% RSLogix 500 project TASTEFULL SELECTIONBINSCRUBBER INDEXER AND UN-STACKER 2-08-2017.RSS, saved by version 10.00.00.00 %
PROJECT "TASTEFUL"    % processor: MicroLogix 1400 %

PROGRAM FILES
  LAD 2 "MAIN"  12 rungs
  LAD 3 "START/MODE"  12 rungs
  LAD 4 "ENCODER"  11 rungs
  LAD 5 "CRADLE"  26 rungs
  LAD 6 "BRUSH"  10 rungs
  LAD 7 "H20 TANKS"  26 rungs
  LAD 8 "AUXILARY"  4 rungs
  LAD 9 "FAULTS"  36 rungs
  LAD 10 "SPARE"  2 rungs
  LAD 11 "STAGING"  8 rungs
  LAD 12 "DESTACK LS"  19 rungs
  LAD 13 "DESTACK"  29 rungs

DATA FILES
  O0 OUTPUT  8 elements
  I1 INPUT  11 elements
  S2 STATUS  66 elements
  B3 BINARY  7 elements
  T4 TIMER  38 elements
  C5 COUNTER  1 elements
  R6 CONTROL  1 elements
  N7 INTEGER  40 elements
  F8 FLOAT  30 elements
  L9   1 elements
  L10   2 elements

LADDER 2 "MAIN"
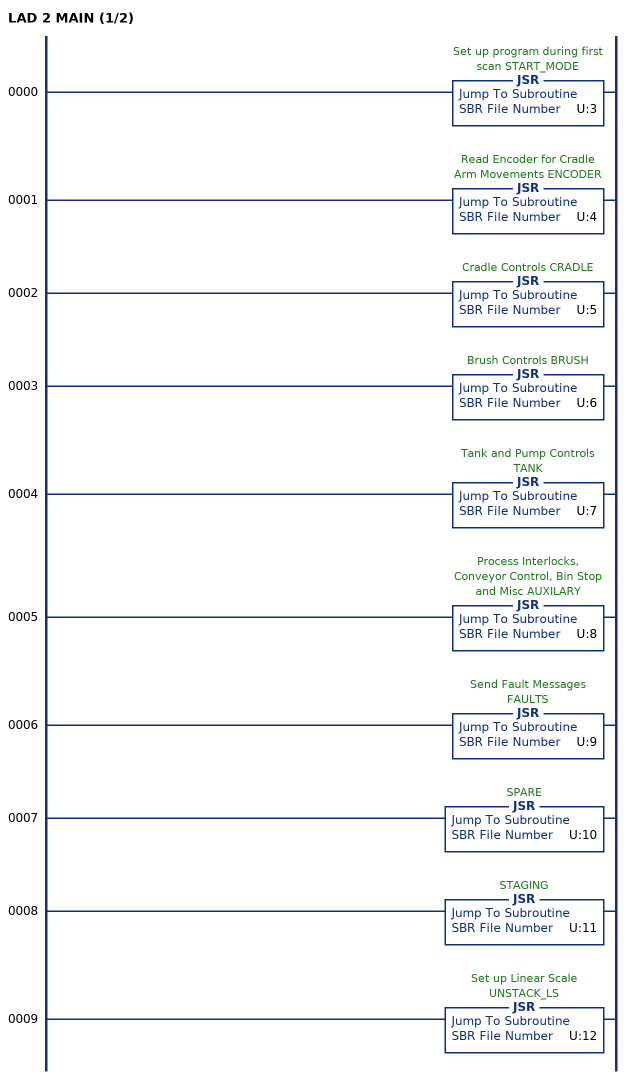
% Rung: 0 %
SOR JSR U:3 EOR
%   U:3  START_MODE  "Set up program during first scan" %
% Rung: 1 %
SOR JSR U:4 EOR
%   U:4  ENCODER  "Read Encoder for Cradle Arm Movements" %
% Rung: 2 %
SOR JSR U:5 EOR
%   U:5  CRADLE  "Cradle Controls" %
% Rung: 3 %
SOR JSR U:6 EOR
%   U:6  BRUSH  "Brush Controls" %
% Rung: 4 %
SOR JSR U:7 EOR
%   U:7  TANK  "Tank and Pump Controls" %
% Rung: 5 %
SOR JSR U:8 EOR
%   U:8  AUXILARY  "Process Interlocks, Conveyor Control, Bin Stop and Misc" %
% Rung: 6 %
SOR JSR U:9 EOR
%   U:9  FAULTS  "Send Fault Messages" %
% Rung: 7 %
SOR JSR U:10 EOR
%   U:10  SPARE %
% Rung: 8 %
SOR JSR U:11 EOR
%   U:11  STAGING %
% Rung: 9 %
SOR JSR U:12 EOR
%   U:12  UNSTACK_LS  "Set up Linear Scale" %

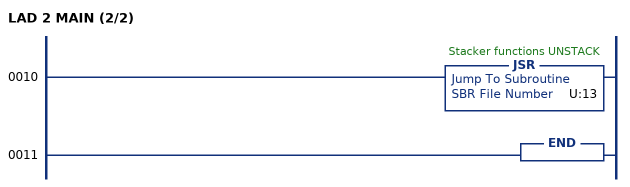
% Rung: 10 %
SOR JSR U:13 EOR
%   U:13  UNSTACK  "Stacker functions" %
% Rung: 11 %
SOR END EOR

LADDER 3 "START/MODE"
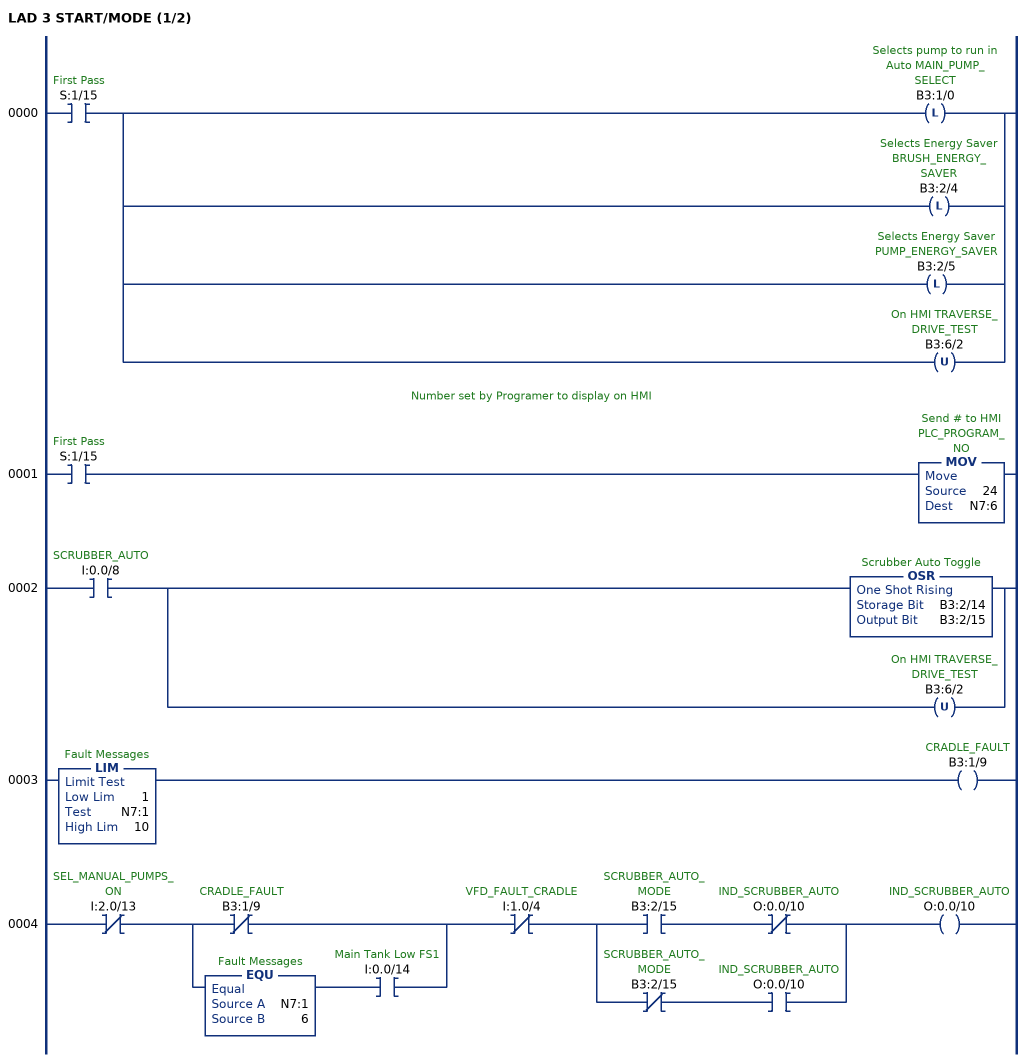
% Rung: 0 %
SOR XIC S:1/15 BST OTL B3:1/0 NXB BST OTL B3:2/4 NXB BST OTL B3:2/5 NXB OTU B3:6/2 BND BND BND EOR
%   S:1/15  "First Pass" %
%   B3:1/0  MAIN_PUMP_SELECT  "Selects pump to run in Auto" %
%   B3:2/4  BRUSH_ENERGY_SAVER  "Selects Energy Saver" %
%   B3:2/5  PUMP_ENERGY_SAVER  "Selects Energy Saver" %
%   B3:6/2  TRAVERSE_DRIVE_TEST  "On HMI" %
% Rung: 1 %
% Number set by Programer to display on HMI %
SOR XIC S:1/15 MOV 24 N7:6 EOR
%   S:1/15  "First Pass" %
%   N7:6  PLC_PROGRAM_NO  "Send # to HMI" %
% Rung: 2 %
SOR XIC I:0.0/8 BST OSR B3:2/14 B3:2/15 NXB OTU B3:6/2 BND EOR
%   I:0.0/8  SCRUBBER_AUTO %
%   B3:2/14  "Scrubber Auto Toggle" %
%   B3:2/15  SCRUBBER_AUTO_MODE %
%   B3:6/2  TRAVERSE_DRIVE_TEST  "On HMI" %
% Rung: 3 %
SOR LIM 1 N7:1 10 OTE B3:1/9 EOR
%   N7:1  "Fault Messages" %
%   B3:1/9  CRADLE_FAULT %
% Rung: 4 %
SOR XIO I:2.0/13 BST XIO B3:1/9 NXB EQU N7:1 6 XIC I:0.0/14 BND XIO I:1.0/4 BST XIC B3:2/15 XIO O:0.0/10 NXB XIO B3:2/15 XIC O:0.0/10 BND OTE O:0.0/10 EOR
%   I:2.0/13  SEL_MANUAL_PUMPS_ON %
%   B3:1/9  CRADLE_FAULT %
%   N7:1  "Fault Messages" %
%   I:0.0/14  FS1  "Main Tank Low" %
%   I:1.0/4  VFD_FAULT_CRADLE %
%   B3:2/15  SCRUBBER_AUTO_MODE %
%   O:0.0/10  IND_SCRUBBER_AUTO %

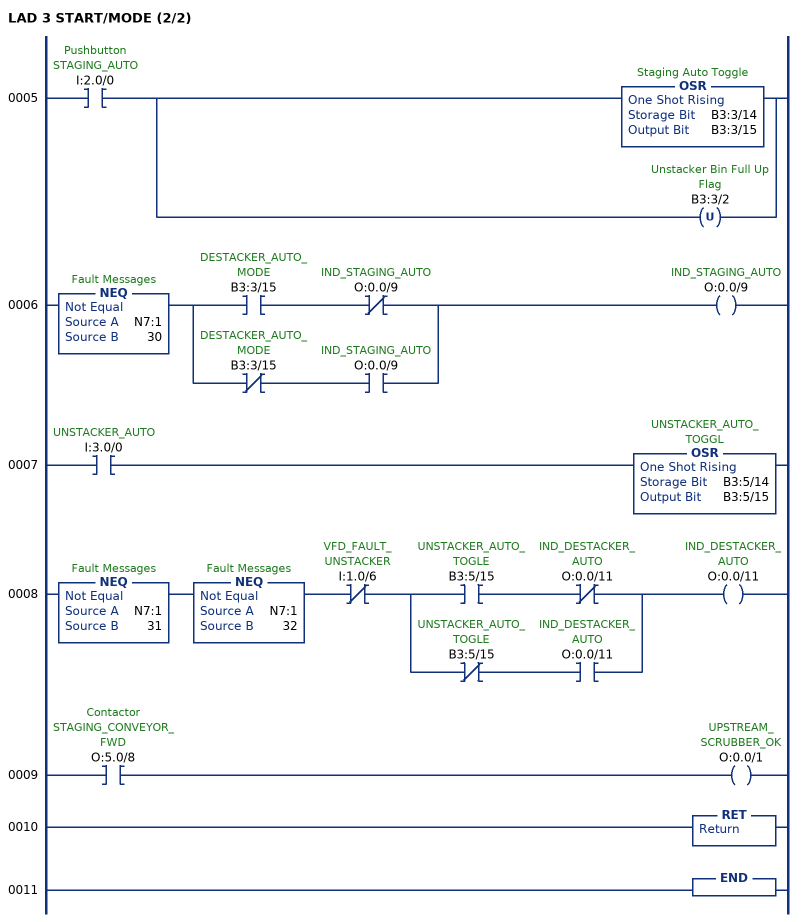
% Rung: 5 %
SOR XIC I:2.0/0 BST OSR B3:3/14 B3:3/15 NXB OTU B3:3/2 BND EOR
%   I:2.0/0  STAGING_AUTO  "Pushbutton" %
%   B3:3/14  "Staging Auto Toggle" %
%   B3:3/15  DESTACKER_AUTO_MODE %
%   B3:3/2  "Unstacker Bin Full Up Flag" %
% Rung: 6 %
SOR NEQ N7:1 30 BST XIC B3:3/15 XIO O:0.0/9 NXB XIO B3:3/15 XIC O:0.0/9 BND OTE O:0.0/9 EOR
%   N7:1  "Fault Messages" %
%   B3:3/15  DESTACKER_AUTO_MODE %
%   O:0.0/9  IND_STAGING_AUTO %
% Rung: 7 %
SOR XIC I:3.0/0 OSR B3:5/14 B3:5/15 EOR
%   I:3.0/0  UNSTACKER_AUTO %
%   B3:5/14  UNSTACKER_AUTO_TOGGL %
%   B3:5/15  UNSTACKER_AUTO_TOGLE %
% Rung: 8 %
SOR NEQ N7:1 31 NEQ N7:1 32 XIO I:1.0/6 BST XIC B3:5/15 XIO O:0.0/11 NXB XIO B3:5/15 XIC O:0.0/11 BND OTE O:0.0/11 EOR
%   N7:1  "Fault Messages" %
%   I:1.0/6  VFD_FAULT_UNSTACKER %
%   B3:5/15  UNSTACKER_AUTO_TOGLE %
%   O:0.0/11  IND_DESTACKER_AUTO %
% Rung: 9 %
SOR XIC O:5.0/8 OTE O:0.0/1 EOR
%   O:5.0/8  STAGING_CONVEYOR_FWD  "Contactor" %
%   O:0.0/1  UPSTREAM_SCRUBBER_OK %
% Rung: 10 %
SOR RET EOR
% Rung: 11 %
SOR END EOR

LADDER 4 "ENCODER"
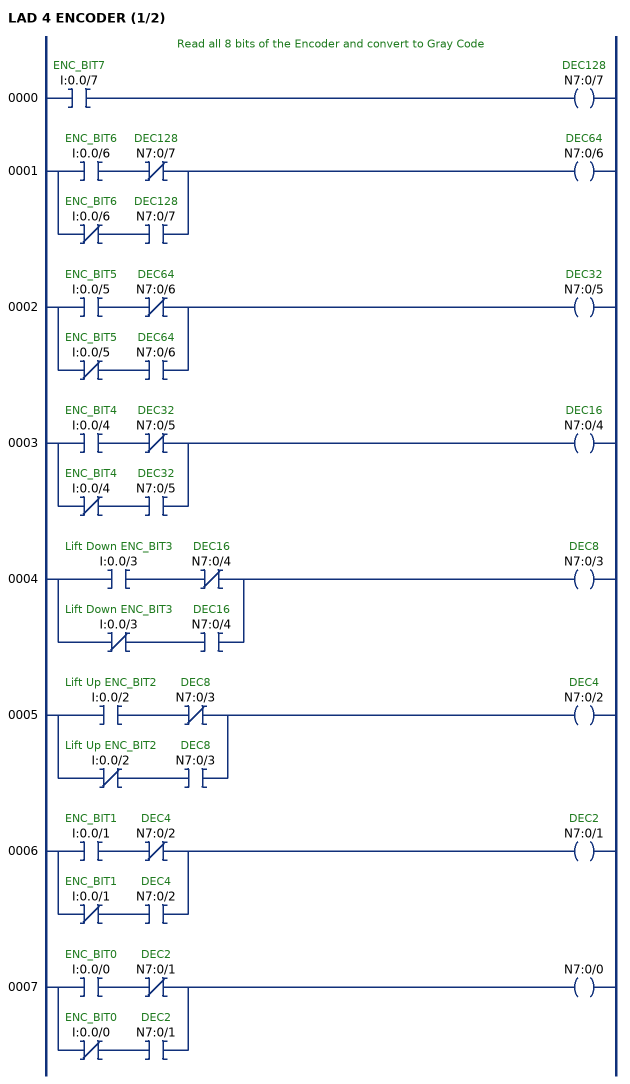
% Rung: 0 %
% Read all 8 bits of the Encoder and convert to Gray Code %
SOR XIC I:0.0/7 OTE N7:0/7 EOR
%   I:0.0/7  ENC_BIT7 %
%   N7:0/7  "DEC128" %
% Rung: 1 %
SOR BST XIC I:0.0/6 XIO N7:0/7 NXB XIO I:0.0/6 XIC N7:0/7 BND OTE N7:0/6 EOR
%   I:0.0/6  ENC_BIT6 %
%   N7:0/7  "DEC128" %
%   N7:0/6  "DEC64" %
% Rung: 2 %
SOR BST XIC I:0.0/5 XIO N7:0/6 NXB XIO I:0.0/5 XIC N7:0/6 BND OTE N7:0/5 EOR
%   I:0.0/5  ENC_BIT5 %
%   N7:0/6  "DEC64" %
%   N7:0/5  "DEC32" %
% Rung: 3 %
SOR BST XIC I:0.0/4 XIO N7:0/5 NXB XIO I:0.0/4 XIC N7:0/5 BND OTE N7:0/4 EOR
%   I:0.0/4  ENC_BIT4 %
%   N7:0/5  "DEC32" %
%   N7:0/4  "DEC16" %
% Rung: 4 %
SOR BST XIC I:0.0/3 XIO N7:0/4 NXB XIO I:0.0/3 XIC N7:0/4 BND OTE N7:0/3 EOR
%   I:0.0/3  ENC_BIT3  "Lift Down" %
%   N7:0/4  "DEC16" %
%   N7:0/3  "DEC8" %
% Rung: 5 %
SOR BST XIC I:0.0/2 XIO N7:0/3 NXB XIO I:0.0/2 XIC N7:0/3 BND OTE N7:0/2 EOR
%   I:0.0/2  ENC_BIT2  "Lift Up" %
%   N7:0/3  "DEC8" %
%   N7:0/2  "DEC4" %
% Rung: 6 %
SOR BST XIC I:0.0/1 XIO N7:0/2 NXB XIO I:0.0/1 XIC N7:0/2 BND OTE N7:0/1 EOR
%   I:0.0/1  ENC_BIT1 %
%   N7:0/2  "DEC4" %
%   N7:0/1  "DEC2" %
% Rung: 7 %
SOR BST XIC I:0.0/0 XIO N7:0/1 NXB XIO I:0.0/0 XIC N7:0/1 BND OTE N7:0/0 EOR
%   I:0.0/0  ENC_BIT0 %
%   N7:0/1  "DEC2" %

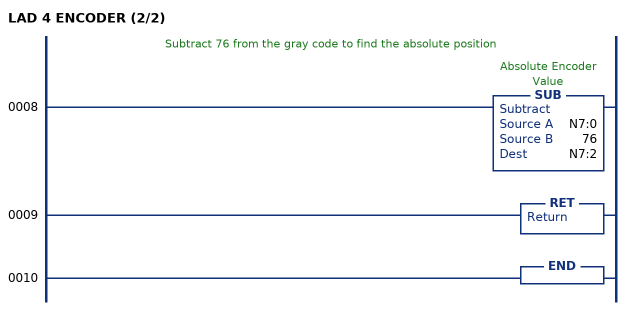
% Rung: 8 %
% Subtract 76 from the gray code to find the absolute position %
SOR SUB N7:0 76 N7:2 EOR
%   N7:0  ENC_POS %
%   N7:2  "Absolute Encoder Value" %
% Rung: 9 %
SOR RET EOR
% Rung: 10 %
SOR END EOR

LADDER 5 "CRADLE"
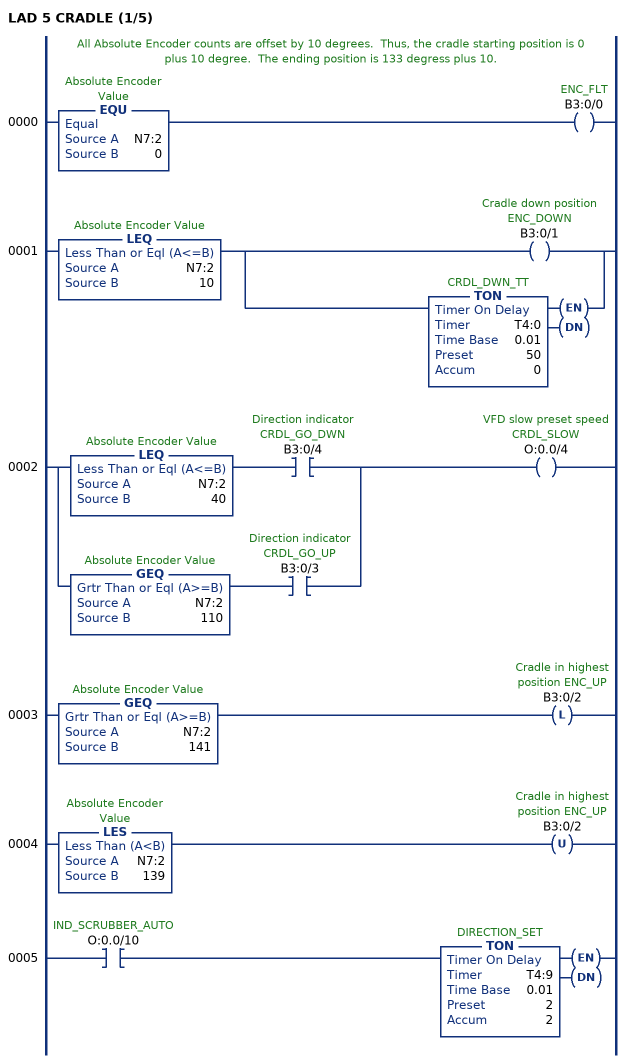
% Rung: 0 %
% All Absolute Encoder counts are offset by 10 degrees.  Thus, the cradle starting position is 0 plus 10 degree.  The ending position is 133 degress plus 10. %
SOR EQU N7:2 0 OTE B3:0/0 EOR
%   N7:2  "Absolute Encoder Value" %
%   B3:0/0  ENC_FLT %
% Rung: 1 %
SOR LEQ N7:2 10 BST OTE B3:0/1 NXB TON T4:0 0.01 50 0 BND EOR
%   N7:2  "Absolute Encoder Value" %
%   B3:0/1  ENC_DOWN  "Cradle down position" %
%   T4:0  CRDL_DWN_TT %
% Rung: 2 %
SOR BST LEQ N7:2 40 XIC B3:0/4 NXB GEQ N7:2 110 XIC B3:0/3 BND OTE O:0.0/4 EOR
%   N7:2  "Absolute Encoder Value" %
%   B3:0/4  CRDL_GO_DWN  "Direction indicator" %
%   B3:0/3  CRDL_GO_UP  "Direction indicator" %
%   O:0.0/4  CRDL_SLOW  "VFD slow preset speed" %
% Rung: 3 %
SOR GEQ N7:2 141 OTL B3:0/2 EOR
%   N7:2  "Absolute Encoder Value" %
%   B3:0/2  ENC_UP  "Cradle in highest position" %
% Rung: 4 %
SOR LES N7:2 139 OTU B3:0/2 EOR
%   N7:2  "Absolute Encoder Value" %
%   B3:0/2  ENC_UP  "Cradle in highest position" %
% Rung: 5 %
SOR XIC O:0.0/10 TON T4:9 0.01 2 2 EOR
%   O:0.0/10  IND_SCRUBBER_AUTO %
%   T4:9  DIRECTION_SET %

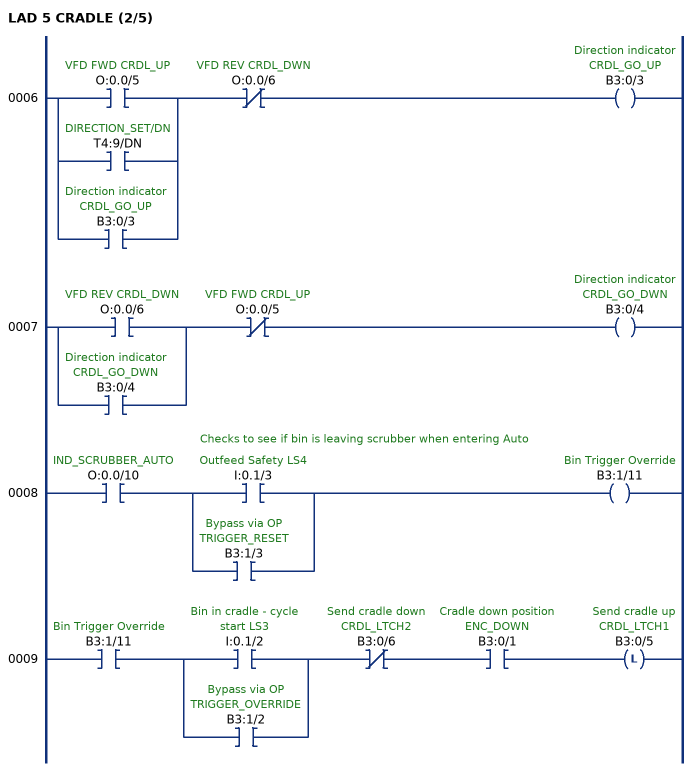
% Rung: 6 %
SOR BST XIC O:0.0/5 NXB XIC T4:9/DN NXB XIC B3:0/3 BND XIO O:0.0/6 OTE B3:0/3 EOR
%   O:0.0/5  CRDL_UP  "VFD FWD" %
%   T4:9  DIRECTION_SET %
%   B3:0/3  CRDL_GO_UP  "Direction indicator" %
%   O:0.0/6  CRDL_DWN  "VFD REV" %
% Rung: 7 %
SOR BST XIC O:0.0/6 NXB XIC B3:0/4 BND XIO O:0.0/5 OTE B3:0/4 EOR
%   O:0.0/6  CRDL_DWN  "VFD REV" %
%   B3:0/4  CRDL_GO_DWN  "Direction indicator" %
%   O:0.0/5  CRDL_UP  "VFD FWD" %
% Rung: 8 %
% Checks to see if bin is leaving scrubber when entering Auto %
SOR XIC O:0.0/10 BST XIC I:0.1/3 NXB XIC B3:1/3 BND OTE B3:1/11 EOR
%   O:0.0/10  IND_SCRUBBER_AUTO %
%   I:0.1/3  LS4  "Outfeed Safety" %
%   B3:1/3  TRIGGER_RESET  "Bypass via OP" %
%   B3:1/11  "Bin Trigger Override" %
% Rung: 9 %
SOR XIC B3:1/11 BST XIC I:0.1/2 NXB XIC B3:1/2 BND XIO B3:0/6 XIC B3:0/1 OTL B3:0/5 EOR
%   B3:1/11  "Bin Trigger Override" %
%   I:0.1/2  LS3  "Bin in cradle - cycle start" %
%   B3:1/2  TRIGGER_OVERRIDE  "Bypass via OP" %
%   B3:0/6  CRDL_LTCH2  "Send cradle down" %
%   B3:0/1  ENC_DOWN  "Cradle down position" %
%   B3:0/5  CRDL_LTCH1  "Send cradle up" %

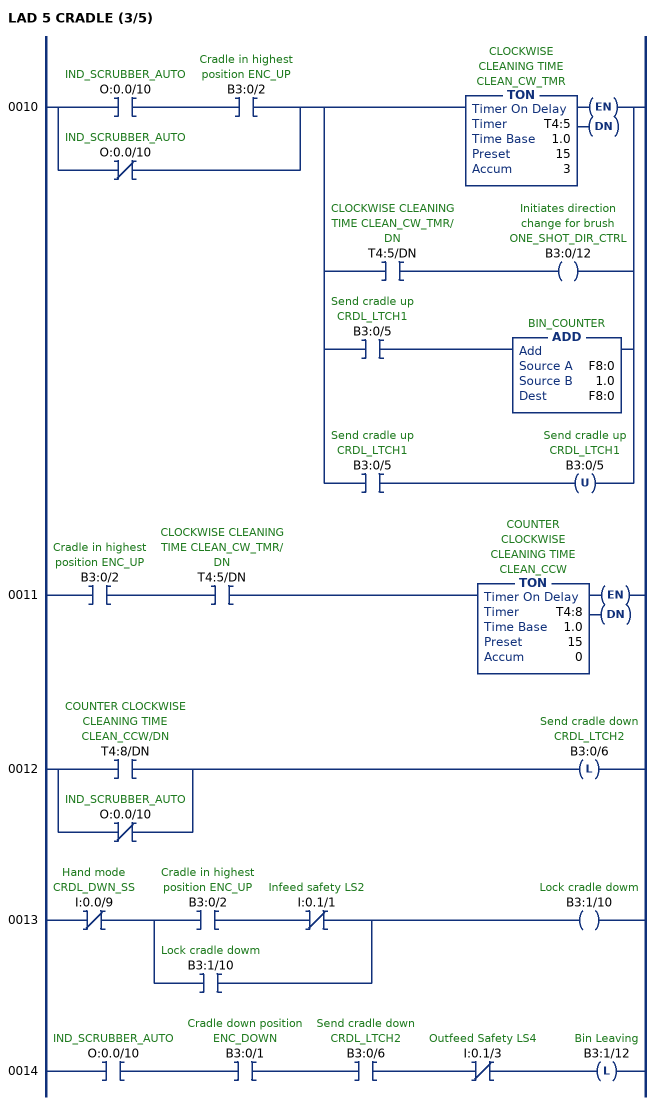
% Rung: 10 %
SOR BST XIC O:0.0/10 XIC B3:0/2 NXB XIO O:0.0/10 BND BST TON T4:5 1.0 15 3 NXB XIC T4:5/DN OTE B3:0/12 NXB BST XIC B3:0/5 ADD F8:0 1.0 F8:0 NXB XIC B3:0/5 OTU B3:0/5 BND BND EOR
%   O:0.0/10  IND_SCRUBBER_AUTO %
%   B3:0/2  ENC_UP  "Cradle in highest position" %
%   T4:5  CLEAN_CW_TMR  "CLOCKWISE CLEANING TIME" %
%   B3:0/12  ONE_SHOT_DIR_CTRL  "Initiates direction change for brush" %
%   B3:0/5  CRDL_LTCH1  "Send cradle up" %
%   F8:0  BIN_COUNTER %
% Rung: 11 %
SOR XIC B3:0/2 XIC T4:5/DN TON T4:8 1.0 15 0 EOR
%   B3:0/2  ENC_UP  "Cradle in highest position" %
%   T4:5  CLEAN_CW_TMR  "CLOCKWISE CLEANING TIME" %
%   T4:8  CLEAN_CCW  "COUNTER CLOCKWISE CLEANING TIME" %
% Rung: 12 %
SOR BST XIC T4:8/DN NXB XIO O:0.0/10 BND OTL B3:0/6 EOR
%   T4:8  CLEAN_CCW  "COUNTER CLOCKWISE CLEANING TIME" %
%   O:0.0/10  IND_SCRUBBER_AUTO %
%   B3:0/6  CRDL_LTCH2  "Send cradle down" %
% Rung: 13 %
SOR XIO I:0.0/9 BST XIC B3:0/2 XIO I:0.1/1 NXB XIC B3:1/10 BND OTE B3:1/10 EOR
%   I:0.0/9  CRDL_DWN_SS  "Hand mode" %
%   B3:0/2  ENC_UP  "Cradle in highest position" %
%   I:0.1/1  LS2  "Infeed safety" %
%   B3:1/10  "Lock cradle dowm" %
% Rung: 14 %
SOR XIC O:0.0/10 XIC B3:0/1 XIC B3:0/6 XIO I:0.1/3 OTL B3:1/12 EOR
%   O:0.0/10  IND_SCRUBBER_AUTO %
%   B3:0/1  ENC_DOWN  "Cradle down position" %
%   B3:0/6  CRDL_LTCH2  "Send cradle down" %
%   I:0.1/3  LS4  "Outfeed Safety" %
%   B3:1/12  "Bin Leaving" %

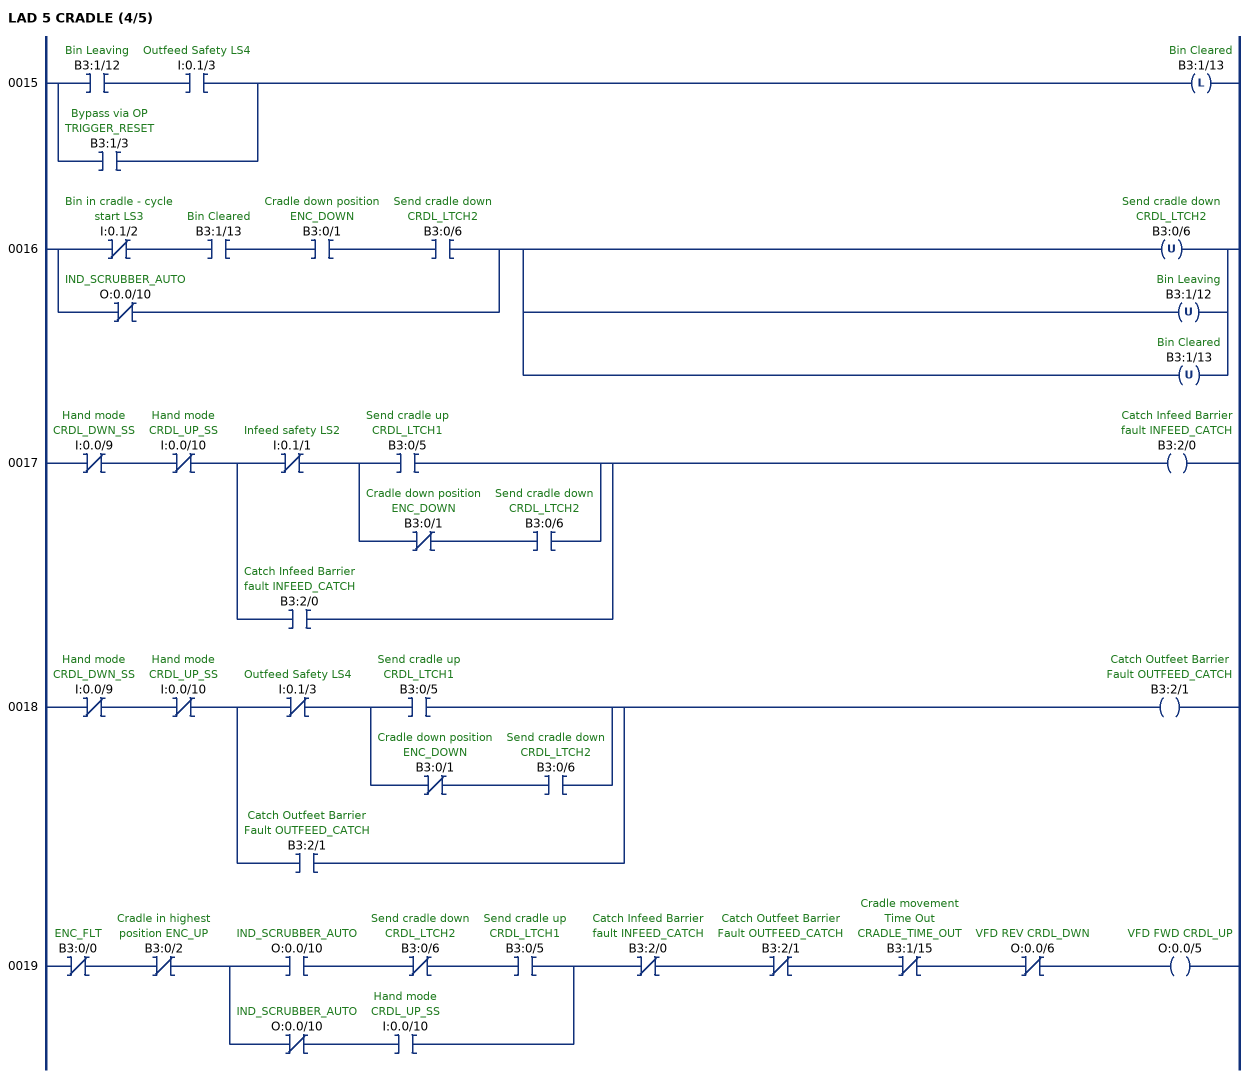
% Rung: 15 %
SOR BST XIC B3:1/12 XIC I:0.1/3 NXB XIC B3:1/3 BND OTL B3:1/13 EOR
%   B3:1/12  "Bin Leaving" %
%   I:0.1/3  LS4  "Outfeed Safety" %
%   B3:1/3  TRIGGER_RESET  "Bypass via OP" %
%   B3:1/13  "Bin Cleared" %
% Rung: 16 %
SOR BST XIO I:0.1/2 XIC B3:1/13 XIC B3:0/1 XIC B3:0/6 NXB XIO O:0.0/10 BND BST OTU B3:0/6 NXB BST OTU B3:1/12 NXB OTU B3:1/13 BND BND EOR
%   I:0.1/2  LS3  "Bin in cradle - cycle start" %
%   B3:1/13  "Bin Cleared" %
%   B3:0/1  ENC_DOWN  "Cradle down position" %
%   B3:0/6  CRDL_LTCH2  "Send cradle down" %
%   O:0.0/10  IND_SCRUBBER_AUTO %
%   B3:1/12  "Bin Leaving" %
% Rung: 17 %
SOR XIO I:0.0/9 XIO I:0.0/10 BST XIO I:0.1/1 BST XIC B3:0/5 NXB XIO B3:0/1 XIC B3:0/6 BND NXB XIC B3:2/0 BND OTE B3:2/0 EOR
%   I:0.0/9  CRDL_DWN_SS  "Hand mode" %
%   I:0.0/10  CRDL_UP_SS  "Hand mode" %
%   I:0.1/1  LS2  "Infeed safety" %
%   B3:0/5  CRDL_LTCH1  "Send cradle up" %
%   B3:0/1  ENC_DOWN  "Cradle down position" %
%   B3:0/6  CRDL_LTCH2  "Send cradle down" %
%   B3:2/0  INFEED_CATCH  "Catch Infeed Barrier fault" %
% Rung: 18 %
SOR XIO I:0.0/9 XIO I:0.0/10 BST XIO I:0.1/3 BST XIC B3:0/5 NXB XIO B3:0/1 XIC B3:0/6 BND NXB XIC B3:2/1 BND OTE B3:2/1 EOR
%   I:0.0/9  CRDL_DWN_SS  "Hand mode" %
%   I:0.0/10  CRDL_UP_SS  "Hand mode" %
%   I:0.1/3  LS4  "Outfeed Safety" %
%   B3:0/5  CRDL_LTCH1  "Send cradle up" %
%   B3:0/1  ENC_DOWN  "Cradle down position" %
%   B3:0/6  CRDL_LTCH2  "Send cradle down" %
%   B3:2/1  OUTFEED_CATCH  "Catch Outfeet Barrier Fault" %
% Rung: 19 %
SOR XIO B3:0/0 XIO B3:0/2 BST XIC O:0.0/10 XIO B3:0/6 XIC B3:0/5 NXB XIO O:0.0/10 XIC I:0.0/10 BND XIO B3:2/0 XIO B3:2/1 XIO B3:1/15 XIO O:0.0/6 OTE O:0.0/5 EOR
%   B3:0/0  ENC_FLT %
%   B3:0/2  ENC_UP  "Cradle in highest position" %
%   O:0.0/10  IND_SCRUBBER_AUTO %
%   B3:0/6  CRDL_LTCH2  "Send cradle down" %
%   B3:0/5  CRDL_LTCH1  "Send cradle up" %
%   I:0.0/10  CRDL_UP_SS  "Hand mode" %
%   B3:2/0  INFEED_CATCH  "Catch Infeed Barrier fault" %
%   B3:2/1  OUTFEED_CATCH  "Catch Outfeet Barrier Fault" %
%   B3:1/15  CRADLE_TIME_OUT  "Cradle movement Time Out" %
%   O:0.0/6  CRDL_DWN  "VFD REV" %
%   O:0.0/5  CRDL_UP  "VFD FWD" %

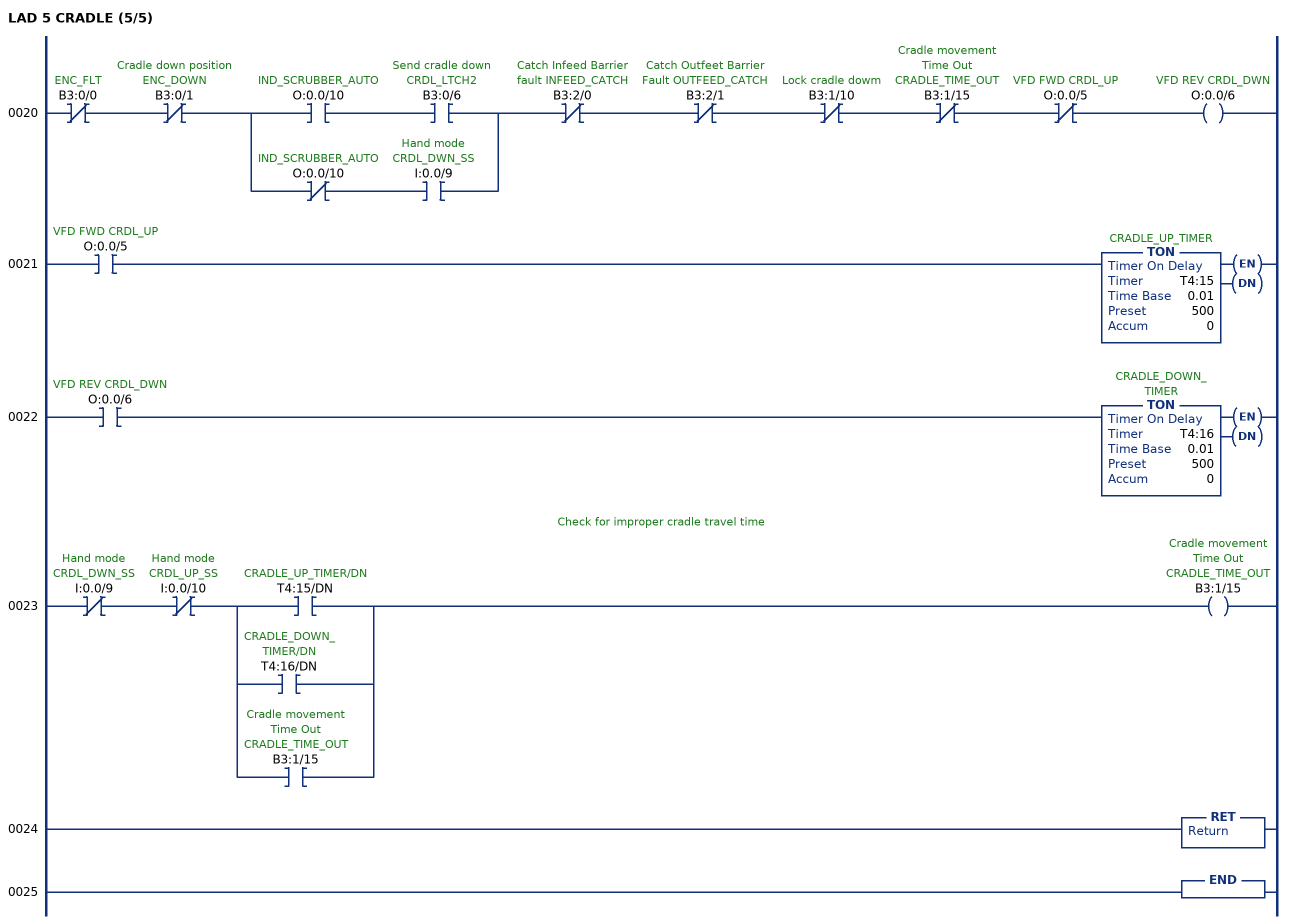
% Rung: 20 %
SOR XIO B3:0/0 XIO B3:0/1 BST XIC O:0.0/10 XIC B3:0/6 NXB XIO O:0.0/10 XIC I:0.0/9 BND XIO B3:2/0 XIO B3:2/1 XIO B3:1/10 XIO B3:1/15 XIO O:0.0/5 OTE O:0.0/6 EOR
%   B3:0/0  ENC_FLT %
%   B3:0/1  ENC_DOWN  "Cradle down position" %
%   O:0.0/10  IND_SCRUBBER_AUTO %
%   B3:0/6  CRDL_LTCH2  "Send cradle down" %
%   I:0.0/9  CRDL_DWN_SS  "Hand mode" %
%   B3:2/0  INFEED_CATCH  "Catch Infeed Barrier fault" %
%   B3:2/1  OUTFEED_CATCH  "Catch Outfeet Barrier Fault" %
%   B3:1/10  "Lock cradle dowm" %
%   B3:1/15  CRADLE_TIME_OUT  "Cradle movement Time Out" %
%   O:0.0/5  CRDL_UP  "VFD FWD" %
%   O:0.0/6  CRDL_DWN  "VFD REV" %
% Rung: 21 %
SOR XIC O:0.0/5 TON T4:15 0.01 500 0 EOR
%   O:0.0/5  CRDL_UP  "VFD FWD" %
%   T4:15  CRADLE_UP_TIMER %
% Rung: 22 %
SOR XIC O:0.0/6 TON T4:16 0.01 500 0 EOR
%   O:0.0/6  CRDL_DWN  "VFD REV" %
%   T4:16  CRADLE_DOWN_TIMER %
% Rung: 23 %
% Check for improper cradle travel time %
SOR XIO I:0.0/9 XIO I:0.0/10 BST BST XIC T4:15/DN NXB XIC T4:16/DN BND NXB XIC B3:1/15 BND OTE B3:1/15 EOR
%   I:0.0/9  CRDL_DWN_SS  "Hand mode" %
%   I:0.0/10  CRDL_UP_SS  "Hand mode" %
%   T4:15  CRADLE_UP_TIMER %
%   T4:16  CRADLE_DOWN_TIMER %
%   B3:1/15  CRADLE_TIME_OUT  "Cradle movement Time Out" %
% Rung: 24 %
SOR RET EOR
% Rung: 25 %
SOR END EOR

LADDER 6 "BRUSH"
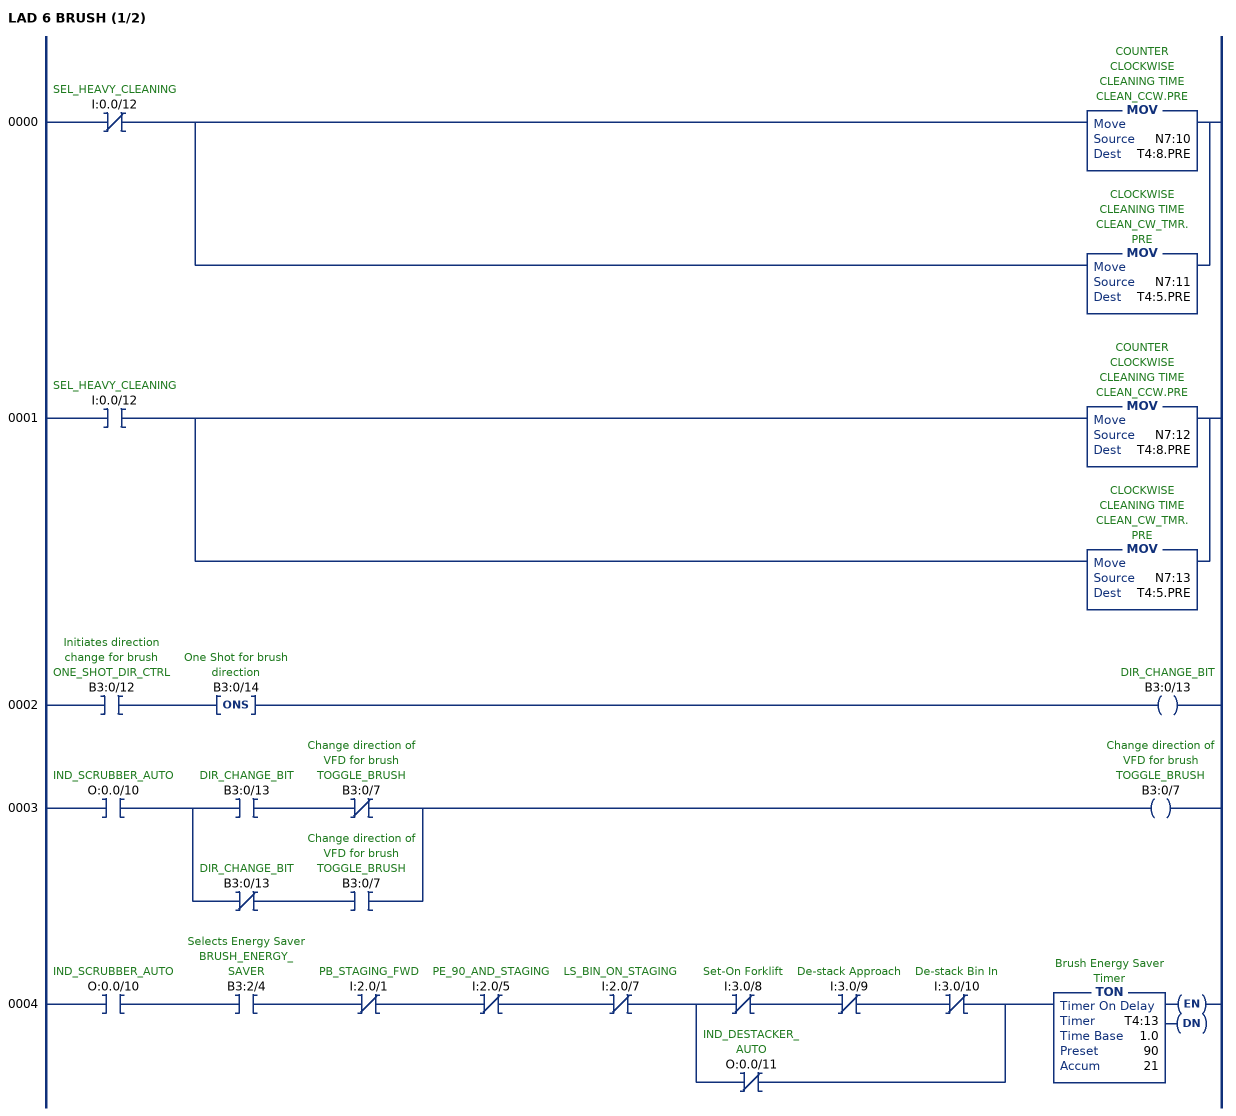
% Rung: 0 %
SOR XIO I:0.0/12 BST MOV N7:10 T4:8.PRE NXB MOV N7:11 T4:5.PRE BND EOR
%   I:0.0/12  SEL_HEAVY_CLEANING %
%   N7:10  NORMAL_CCW_TIME %
%   T4:8  CLEAN_CCW  "COUNTER CLOCKWISE CLEANING TIME" %
%   N7:11  NORMAL_CW_CLEANING %
%   T4:5  CLEAN_CW_TMR  "CLOCKWISE CLEANING TIME" %
% Rung: 1 %
SOR XIC I:0.0/12 BST MOV N7:12 T4:8.PRE NXB MOV N7:13 T4:5.PRE BND EOR
%   I:0.0/12  SEL_HEAVY_CLEANING %
%   N7:12  HEAVY_CCW_CLEANING %
%   T4:8  CLEAN_CCW  "COUNTER CLOCKWISE CLEANING TIME" %
%   N7:13  HEAVY_CW_CLEANING %
%   T4:5  CLEAN_CW_TMR  "CLOCKWISE CLEANING TIME" %
% Rung: 2 %
SOR XIC B3:0/12 ONS B3:0/14 OTE B3:0/13 EOR
%   B3:0/12  ONE_SHOT_DIR_CTRL  "Initiates direction change for brush" %
%   B3:0/14  "One Shot for brush direction" %
%   B3:0/13  DIR_CHANGE_BIT %
% Rung: 3 %
SOR XIC O:0.0/10 BST XIC B3:0/13 XIO B3:0/7 NXB XIO B3:0/13 XIC B3:0/7 BND OTE B3:0/7 EOR
%   O:0.0/10  IND_SCRUBBER_AUTO %
%   B3:0/13  DIR_CHANGE_BIT %
%   B3:0/7  TOGGLE_BRUSH  "Change direction of VFD for brush" %
% Rung: 4 %
SOR XIC O:0.0/10 XIC B3:2/4 XIO I:2.0/1 XIO I:2.0/5 XIO I:2.0/7 BST XIO I:3.0/8 XIO I:3.0/9 XIO I:3.0/10 NXB XIO O:0.0/11 BND TON T4:13 1.0 90 21 EOR
%   O:0.0/10  IND_SCRUBBER_AUTO %
%   B3:2/4  BRUSH_ENERGY_SAVER  "Selects Energy Saver" %
%   I:2.0/1  PB_STAGING_FWD %
%   I:2.0/5  PE_90_AND_STAGING %
%   I:2.0/7  LS_BIN_ON_STAGING %
%   I:3.0/8  "Set-On Forklift" %
%   I:3.0/9  "De-stack Approach" %
%   I:3.0/10  "De-stack Bin In" %
%   O:0.0/11  IND_DESTACKER_AUTO %
%   T4:13  "Brush Energy Saver Timer" %

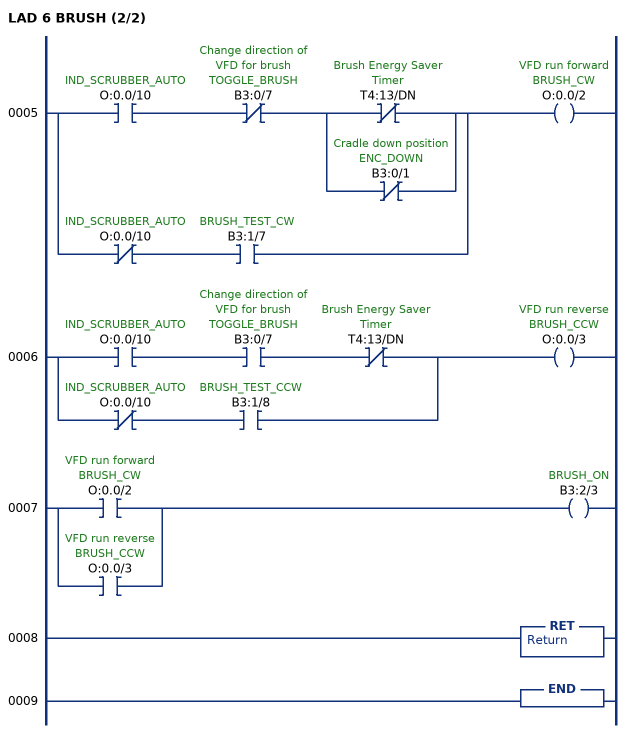
% Rung: 5 %
SOR BST XIC O:0.0/10 XIO B3:0/7 BST XIO T4:13/DN NXB XIO B3:0/1 BND NXB XIO O:0.0/10 XIC B3:1/7 BND OTE O:0.0/2 EOR
%   O:0.0/10  IND_SCRUBBER_AUTO %
%   B3:0/7  TOGGLE_BRUSH  "Change direction of VFD for brush" %
%   T4:13  "Brush Energy Saver Timer" %
%   B3:0/1  ENC_DOWN  "Cradle down position" %
%   B3:1/7  BRUSH_TEST_CW %
%   O:0.0/2  BRUSH_CW  "VFD run forward" %
% Rung: 6 %
SOR BST XIC O:0.0/10 XIC B3:0/7 XIO T4:13/DN NXB XIO O:0.0/10 XIC B3:1/8 BND OTE O:0.0/3 EOR
%   O:0.0/10  IND_SCRUBBER_AUTO %
%   B3:0/7  TOGGLE_BRUSH  "Change direction of VFD for brush" %
%   T4:13  "Brush Energy Saver Timer" %
%   B3:1/8  BRUSH_TEST_CCW %
%   O:0.0/3  BRUSH_CCW  "VFD run reverse" %
% Rung: 7 %
SOR BST XIC O:0.0/2 NXB XIC O:0.0/3 BND OTE B3:2/3 EOR
%   O:0.0/2  BRUSH_CW  "VFD run forward" %
%   O:0.0/3  BRUSH_CCW  "VFD run reverse" %
%   B3:2/3  BRUSH_ON %
% Rung: 8 %
SOR RET EOR
% Rung: 9 %
SOR END EOR

LADDER 7 "H20 TANKS"
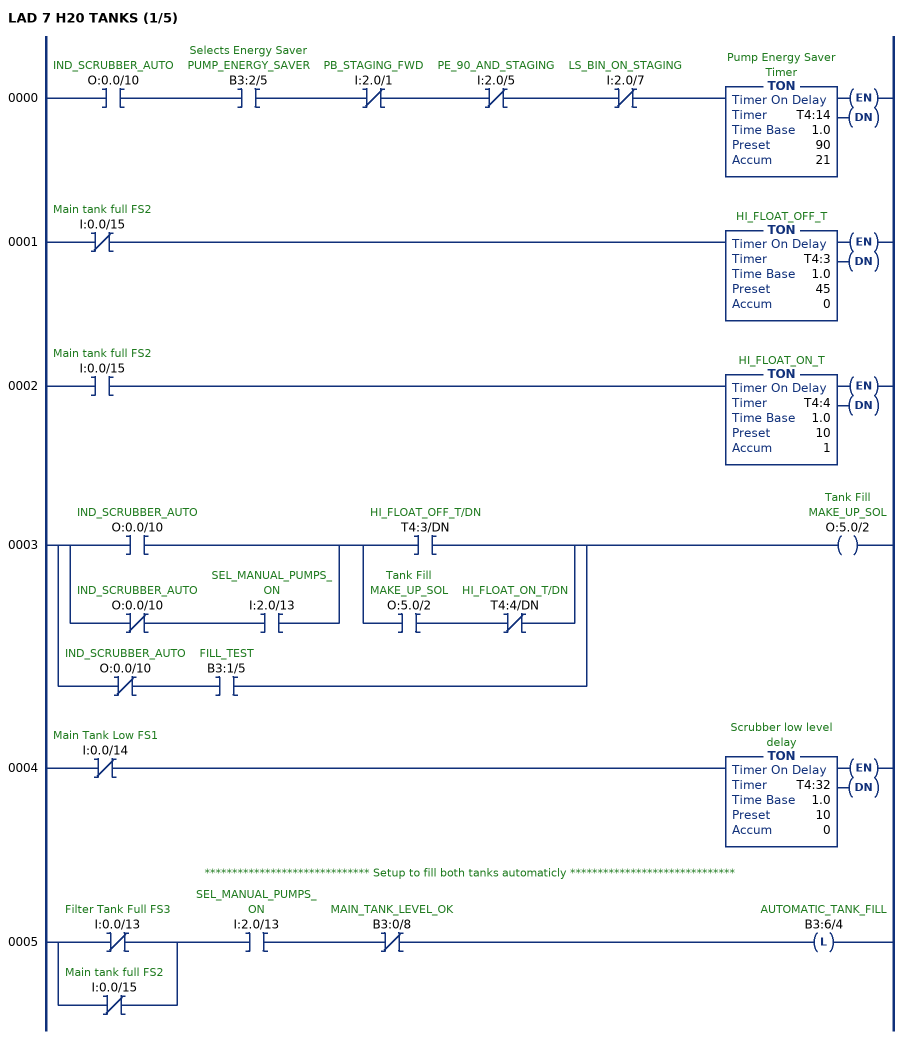
% Rung: 0 %
SOR XIC O:0.0/10 XIC B3:2/5 XIO I:2.0/1 XIO I:2.0/5 XIO I:2.0/7 TON T4:14 1.0 90 21 EOR
%   O:0.0/10  IND_SCRUBBER_AUTO %
%   B3:2/5  PUMP_ENERGY_SAVER  "Selects Energy Saver" %
%   I:2.0/1  PB_STAGING_FWD %
%   I:2.0/5  PE_90_AND_STAGING %
%   I:2.0/7  LS_BIN_ON_STAGING %
%   T4:14  "Pump Energy Saver Timer" %
% Rung: 1 %
SOR XIO I:0.0/15 TON T4:3 1.0 45 0 EOR
%   I:0.0/15  FS2  "Main tank full" %
%   T4:3  HI_FLOAT_OFF_T %
% Rung: 2 %
SOR XIC I:0.0/15 TON T4:4 1.0 10 1 EOR
%   I:0.0/15  FS2  "Main tank full" %
%   T4:4  HI_FLOAT_ON_T %
% Rung: 3 %
SOR BST BST XIC O:0.0/10 NXB XIO O:0.0/10 XIC I:2.0/13 BND BST XIC T4:3/DN NXB XIC O:5.0/2 XIO T4:4/DN BND NXB XIO O:0.0/10 XIC B3:1/5 BND OTE O:5.0/2 EOR
%   O:0.0/10  IND_SCRUBBER_AUTO %
%   I:2.0/13  SEL_MANUAL_PUMPS_ON %
%   T4:3  HI_FLOAT_OFF_T %
%   O:5.0/2  MAKE_UP_SOL  "Tank Fill" %
%   T4:4  HI_FLOAT_ON_T %
%   B3:1/5  FILL_TEST %
% Rung: 4 %
SOR XIO I:0.0/14 TON T4:32 1.0 10 0 EOR
%   I:0.0/14  FS1  "Main Tank Low" %
%   T4:32  "Scrubber low level delay" %
% Rung: 5 %
% ****************************** Setup to fill both tanks automaticly ****************************** %
SOR BST XIO I:0.0/13 NXB XIO I:0.0/15 BND XIC I:2.0/13 XIO B3:0/8 OTL B3:6/4 EOR
%   I:0.0/13  FS3  "Filter Tank Full" %
%   I:0.0/15  FS2  "Main tank full" %
%   I:2.0/13  SEL_MANUAL_PUMPS_ON %
%   B3:0/8  MAIN_TANK_LEVEL_OK %
%   B3:6/4  AUTOMATIC_TANK_FILL %

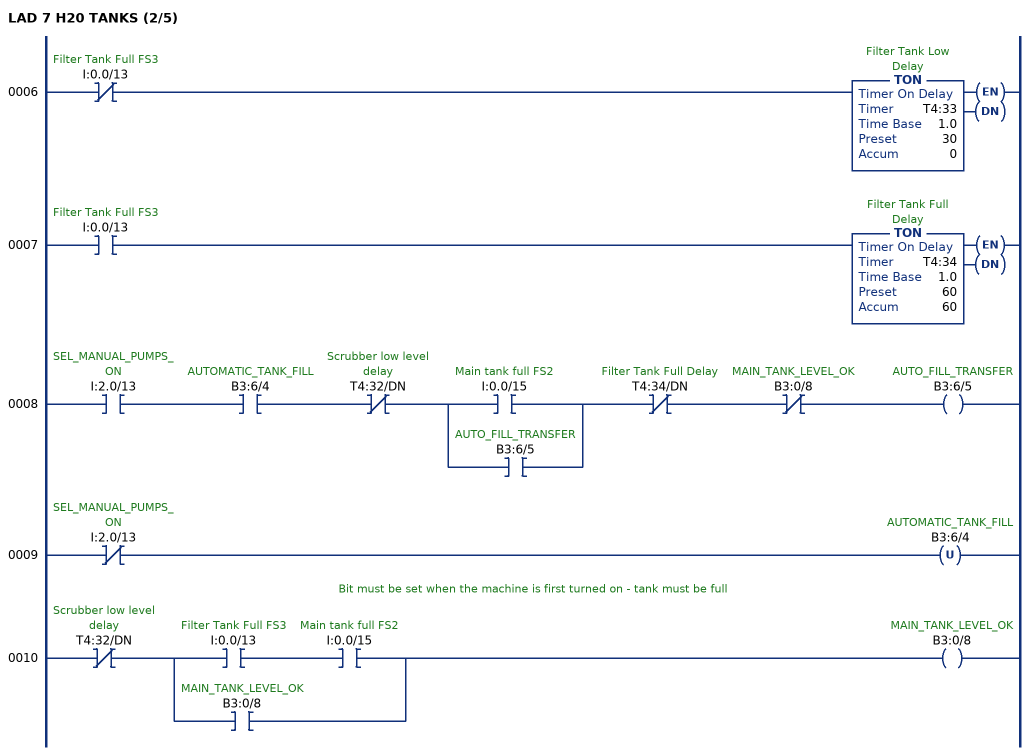
% Rung: 6 %
SOR XIO I:0.0/13 TON T4:33 1.0 30 0 EOR
%   I:0.0/13  FS3  "Filter Tank Full" %
%   T4:33  "Filter Tank Low Delay" %
% Rung: 7 %
SOR XIC I:0.0/13 TON T4:34 1.0 60 60 EOR
%   I:0.0/13  FS3  "Filter Tank Full" %
%   T4:34  "Filter Tank Full Delay" %
% Rung: 8 %
SOR XIC I:2.0/13 XIC B3:6/4 XIO T4:32/DN BST XIC I:0.0/15 NXB XIC B3:6/5 BND XIO T4:34/DN XIO B3:0/8 OTE B3:6/5 EOR
%   I:2.0/13  SEL_MANUAL_PUMPS_ON %
%   B3:6/4  AUTOMATIC_TANK_FILL %
%   T4:32  "Scrubber low level delay" %
%   I:0.0/15  FS2  "Main tank full" %
%   B3:6/5  AUTO_FILL_TRANSFER %
%   T4:34  "Filter Tank Full Delay" %
%   B3:0/8  MAIN_TANK_LEVEL_OK %
% Rung: 9 %
SOR XIO I:2.0/13 OTU B3:6/4 EOR
%   I:2.0/13  SEL_MANUAL_PUMPS_ON %
%   B3:6/4  AUTOMATIC_TANK_FILL %
% Rung: 10 %
% Bit must be set when the machine is first turned on - tank must be full %
SOR XIO T4:32/DN BST XIC I:0.0/13 XIC I:0.0/15 NXB XIC B3:0/8 BND OTE B3:0/8 EOR
%   T4:32  "Scrubber low level delay" %
%   I:0.0/13  FS3  "Filter Tank Full" %
%   I:0.0/15  FS2  "Main tank full" %
%   B3:0/8  MAIN_TANK_LEVEL_OK %

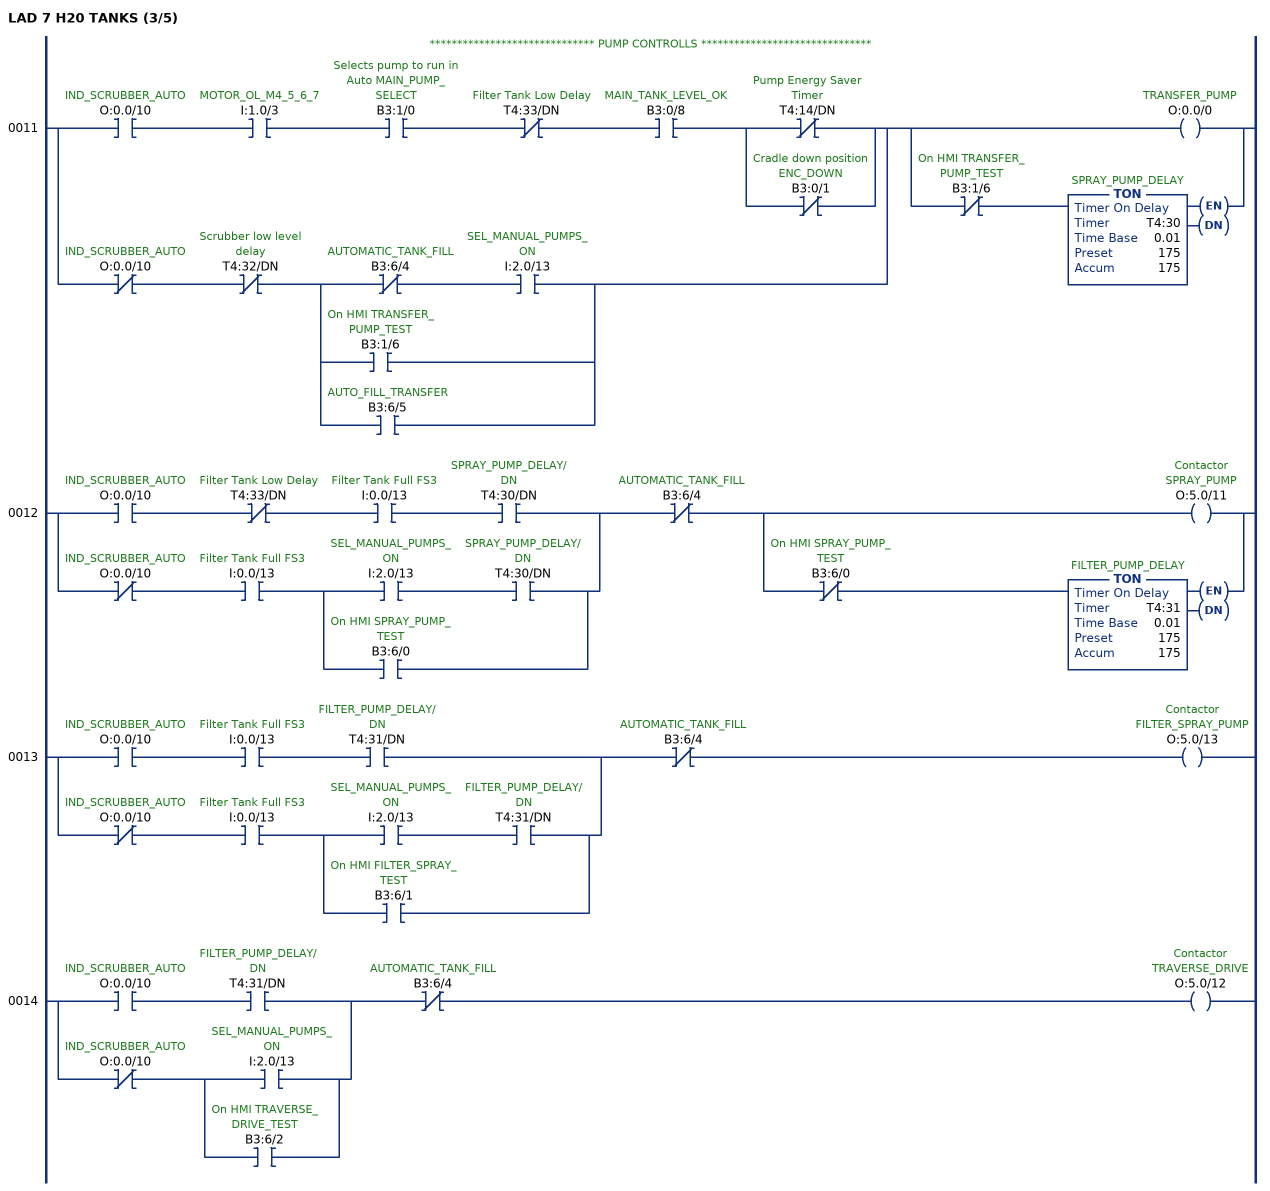
% Rung: 11 %
% ****************************** PUMP CONTROLLS ******************************* %
SOR BST XIC O:0.0/10 XIC I:1.0/3 XIC B3:1/0 XIO T4:33/DN XIC B3:0/8 BST XIO T4:14/DN NXB XIO B3:0/1 BND NXB XIO O:0.0/10 XIO T4:32/DN BST XIO B3:6/4 XIC I:2.0/13 NXB BST XIC B3:1/6 NXB XIC B3:6/5 BND BND BND BST OTE O:0.0/0 NXB XIO B3:1/6 TON T4:30 0.01 175 175 BND EOR
%   O:0.0/10  IND_SCRUBBER_AUTO %
%   I:1.0/3  MOTOR_OL_M4_5_6_7 %
%   B3:1/0  MAIN_PUMP_SELECT  "Selects pump to run in Auto" %
%   T4:33  "Filter Tank Low Delay" %
%   B3:0/8  MAIN_TANK_LEVEL_OK %
%   T4:14  "Pump Energy Saver Timer" %
%   B3:0/1  ENC_DOWN  "Cradle down position" %
%   T4:32  "Scrubber low level delay" %
%   B3:6/4  AUTOMATIC_TANK_FILL %
%   I:2.0/13  SEL_MANUAL_PUMPS_ON %
%   B3:1/6  TRANSFER_PUMP_TEST  "On HMI" %
%   B3:6/5  AUTO_FILL_TRANSFER %
%   O:0.0/0  TRANSFER_PUMP %
%   T4:30  SPRAY_PUMP_DELAY %
% Rung: 12 %
SOR BST XIC O:0.0/10 XIO T4:33/DN XIC I:0.0/13 XIC T4:30/DN NXB XIO O:0.0/10 XIC I:0.0/13 BST XIC I:2.0/13 XIC T4:30/DN NXB XIC B3:6/0 BND BND XIO B3:6/4 BST OTE O:5.0/11 NXB XIO B3:6/0 TON T4:31 0.01 175 175 BND EOR
%   O:0.0/10  IND_SCRUBBER_AUTO %
%   T4:33  "Filter Tank Low Delay" %
%   I:0.0/13  FS3  "Filter Tank Full" %
%   T4:30  SPRAY_PUMP_DELAY %
%   I:2.0/13  SEL_MANUAL_PUMPS_ON %
%   B3:6/0  SPRAY_PUMP_TEST  "On HMI" %
%   B3:6/4  AUTOMATIC_TANK_FILL %
%   O:5.0/11  SPRAY_PUMP  "Contactor" %
%   T4:31  FILTER_PUMP_DELAY %
% Rung: 13 %
SOR BST XIC O:0.0/10 XIC I:0.0/13 XIC T4:31/DN NXB XIO O:0.0/10 XIC I:0.0/13 BST XIC I:2.0/13 XIC T4:31/DN NXB XIC B3:6/1 BND BND XIO B3:6/4 OTE O:5.0/13 EOR
%   O:0.0/10  IND_SCRUBBER_AUTO %
%   I:0.0/13  FS3  "Filter Tank Full" %
%   T4:31  FILTER_PUMP_DELAY %
%   I:2.0/13  SEL_MANUAL_PUMPS_ON %
%   B3:6/1  FILTER_SPRAY_TEST  "On HMI" %
%   B3:6/4  AUTOMATIC_TANK_FILL %
%   O:5.0/13  FILTER_SPRAY_PUMP  "Contactor" %
% Rung: 14 %
SOR BST XIC O:0.0/10 XIC T4:31/DN NXB XIO O:0.0/10 BST XIC I:2.0/13 NXB XIC B3:6/2 BND BND XIO B3:6/4 OTE O:5.0/12 EOR
%   O:0.0/10  IND_SCRUBBER_AUTO %
%   T4:31  FILTER_PUMP_DELAY %
%   I:2.0/13  SEL_MANUAL_PUMPS_ON %
%   B3:6/2  TRAVERSE_DRIVE_TEST  "On HMI" %
%   B3:6/4  AUTOMATIC_TANK_FILL %
%   O:5.0/12  TRAVERSE_DRIVE  "Contactor" %

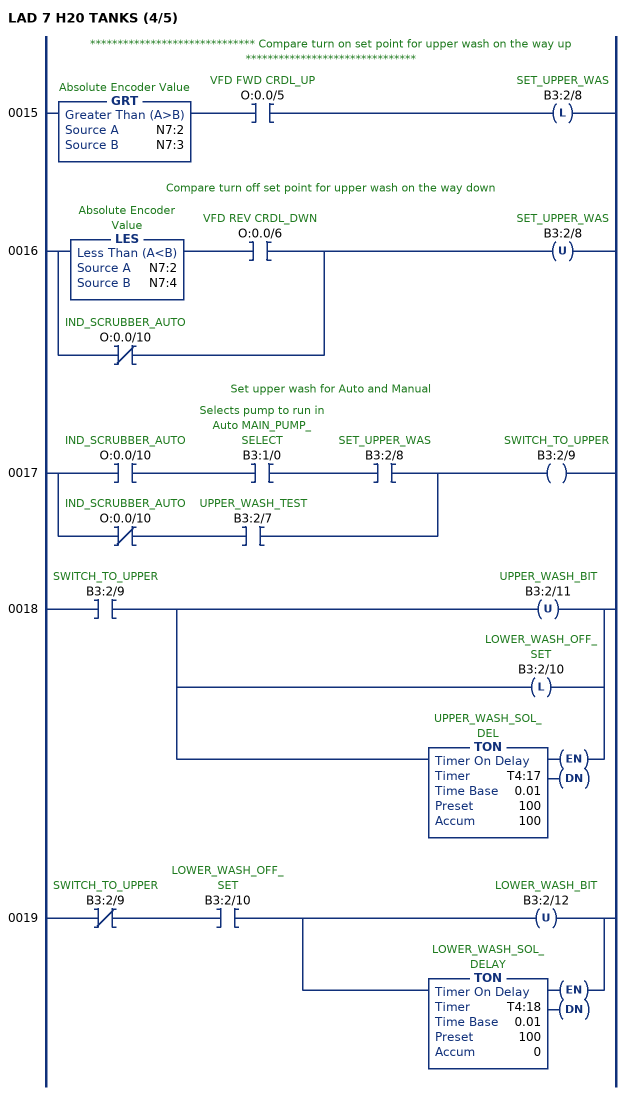
% Rung: 15 %
% ****************************** Compare turn on set point for upper wash on the way up ******************************* %
SOR GRT N7:2 N7:3 XIC O:0.0/5 OTL B3:2/8 EOR
%   N7:2  "Absolute Encoder Value" %
%   N7:3  UPPER_WASH_TURN_ON %
%   O:0.0/5  CRDL_UP  "VFD FWD" %
%   B3:2/8  SET_UPPER_WAS %
% Rung: 16 %
% Compare turn off set point for upper wash on the way down %
SOR BST LES N7:2 N7:4 XIC O:0.0/6 NXB XIO O:0.0/10 BND OTU B3:2/8 EOR
%   N7:2  "Absolute Encoder Value" %
%   N7:4  UPPER_WASH_TURN_OFF %
%   O:0.0/6  CRDL_DWN  "VFD REV" %
%   O:0.0/10  IND_SCRUBBER_AUTO %
%   B3:2/8  SET_UPPER_WAS %
% Rung: 17 %
% Set upper wash for Auto and Manual %
SOR BST XIC O:0.0/10 XIC B3:1/0 XIC B3:2/8 NXB XIO O:0.0/10 XIC B3:2/7 BND OTE B3:2/9 EOR
%   O:0.0/10  IND_SCRUBBER_AUTO %
%   B3:1/0  MAIN_PUMP_SELECT  "Selects pump to run in Auto" %
%   B3:2/8  SET_UPPER_WAS %
%   B3:2/7  UPPER_WASH_TEST %
%   B3:2/9  SWITCH_TO_UPPER %
% Rung: 18 %
SOR XIC B3:2/9 BST OTU B3:2/11 NXB BST OTL B3:2/10 NXB TON T4:17 0.01 100 100 BND BND EOR
%   B3:2/9  SWITCH_TO_UPPER %
%   B3:2/11  UPPER_WASH_BIT %
%   B3:2/10  LOWER_WASH_OFF_SET %
%   T4:17  UPPER_WASH_SOL_DEL %
% Rung: 19 %
SOR XIO B3:2/9 XIC B3:2/10 BST OTU B3:2/12 NXB TON T4:18 0.01 100 0 BND EOR
%   B3:2/9  SWITCH_TO_UPPER %
%   B3:2/10  LOWER_WASH_OFF_SET %
%   B3:2/12  LOWER_WASH_BIT %
%   T4:18  LOWER_WASH_SOL_DELAY %

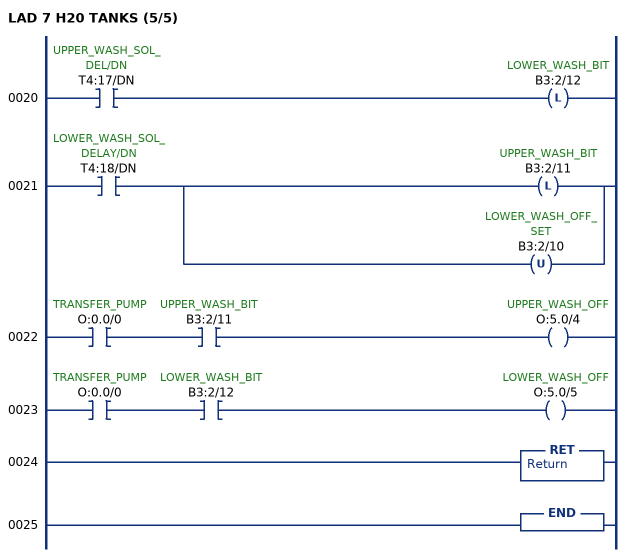
% Rung: 20 %
SOR XIC T4:17/DN OTL B3:2/12 EOR
%   T4:17  UPPER_WASH_SOL_DEL %
%   B3:2/12  LOWER_WASH_BIT %
% Rung: 21 %
SOR XIC T4:18/DN BST OTL B3:2/11 NXB OTU B3:2/10 BND EOR
%   T4:18  LOWER_WASH_SOL_DELAY %
%   B3:2/11  UPPER_WASH_BIT %
%   B3:2/10  LOWER_WASH_OFF_SET %
% Rung: 22 %
SOR XIC O:0.0/0 XIC B3:2/11 OTE O:5.0/4 EOR
%   O:0.0/0  TRANSFER_PUMP %
%   B3:2/11  UPPER_WASH_BIT %
%   O:5.0/4  UPPER_WASH_OFF %
% Rung: 23 %
SOR XIC O:0.0/0 XIC B3:2/12 OTE O:5.0/5 EOR
%   O:0.0/0  TRANSFER_PUMP %
%   B3:2/12  LOWER_WASH_BIT %
%   O:5.0/5  LOWER_WASH_OFF %
% Rung: 24 %
SOR RET EOR
% Rung: 25 %
SOR END EOR

LADDER 8 "AUXILARY"
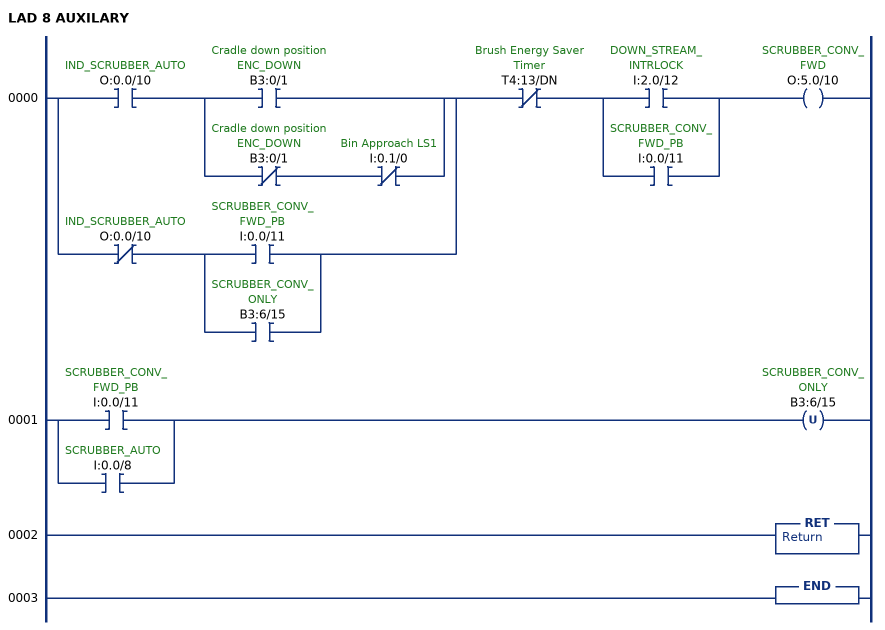
% Rung: 0 %
SOR BST XIC O:0.0/10 BST XIC B3:0/1 NXB XIO B3:0/1 XIO I:0.1/0 BND NXB XIO O:0.0/10 BST XIC I:0.0/11 NXB XIC B3:6/15 BND BND XIO T4:13/DN BST XIC I:2.0/12 NXB XIC I:0.0/11 BND OTE O:5.0/10 EOR
%   O:0.0/10  IND_SCRUBBER_AUTO %
%   B3:0/1  ENC_DOWN  "Cradle down position" %
%   I:0.1/0  LS1  "Bin Approach" %
%   I:0.0/11  SCRUBBER_CONV_FWD_PB %
%   B3:6/15  SCRUBBER_CONV_ONLY %
%   T4:13  "Brush Energy Saver Timer" %
%   I:2.0/12  DOWN_STREAM_INTRLOCK %
%   O:5.0/10  SCRUBBER_CONV_FWD %
% Rung: 1 %
SOR BST XIC I:0.0/11 NXB XIC I:0.0/8 BND OTU B3:6/15 EOR
%   I:0.0/11  SCRUBBER_CONV_FWD_PB %
%   I:0.0/8  SCRUBBER_AUTO %
%   B3:6/15  SCRUBBER_CONV_ONLY %
% Rung: 2 %
SOR RET EOR
% Rung: 3 %
SOR END EOR

LADDER 9 "FAULTS"
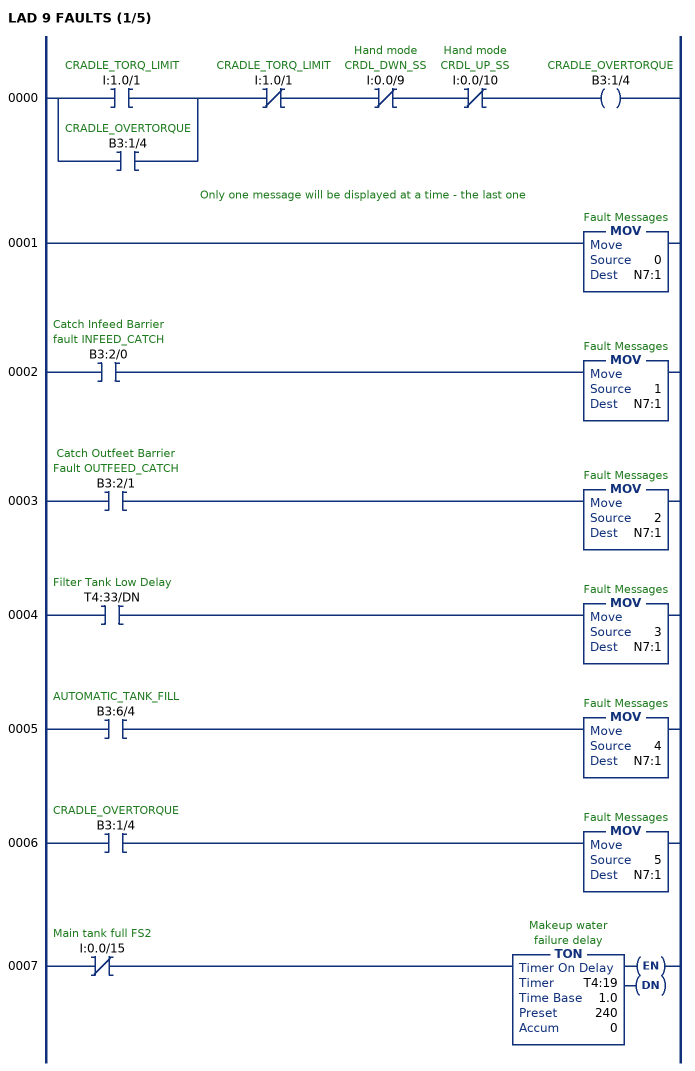
% Rung: 0 %
SOR BST XIC I:1.0/1 NXB XIC B3:1/4 BND XIO I:1.0/1 XIO I:0.0/9 XIO I:0.0/10 OTE B3:1/4 EOR
%   I:1.0/1  CRADLE_TORQ_LIMIT %
%   B3:1/4  CRADLE_OVERTORQUE %
%   I:0.0/9  CRDL_DWN_SS  "Hand mode" %
%   I:0.0/10  CRDL_UP_SS  "Hand mode" %
% Rung: 1 %
% Only one message will be displayed at a time - the last one %
SOR MOV 0 N7:1 EOR
%   N7:1  "Fault Messages" %
% Rung: 2 %
SOR XIC B3:2/0 MOV 1 N7:1 EOR
%   B3:2/0  INFEED_CATCH  "Catch Infeed Barrier fault" %
%   N7:1  "Fault Messages" %
% Rung: 3 %
SOR XIC B3:2/1 MOV 2 N7:1 EOR
%   B3:2/1  OUTFEED_CATCH  "Catch Outfeet Barrier Fault" %
%   N7:1  "Fault Messages" %
% Rung: 4 %
SOR XIC T4:33/DN MOV 3 N7:1 EOR
%   T4:33  "Filter Tank Low Delay" %
%   N7:1  "Fault Messages" %
% Rung: 5 %
SOR XIC B3:6/4 MOV 4 N7:1 EOR
%   B3:6/4  AUTOMATIC_TANK_FILL %
%   N7:1  "Fault Messages" %
% Rung: 6 %
SOR XIC B3:1/4 MOV 5 N7:1 EOR
%   B3:1/4  CRADLE_OVERTORQUE %
%   N7:1  "Fault Messages" %
% Rung: 7 %
SOR XIO I:0.0/15 TON T4:19 1.0 240 0 EOR
%   I:0.0/15  FS2  "Main tank full" %
%   T4:19  "Makeup water failure delay" %

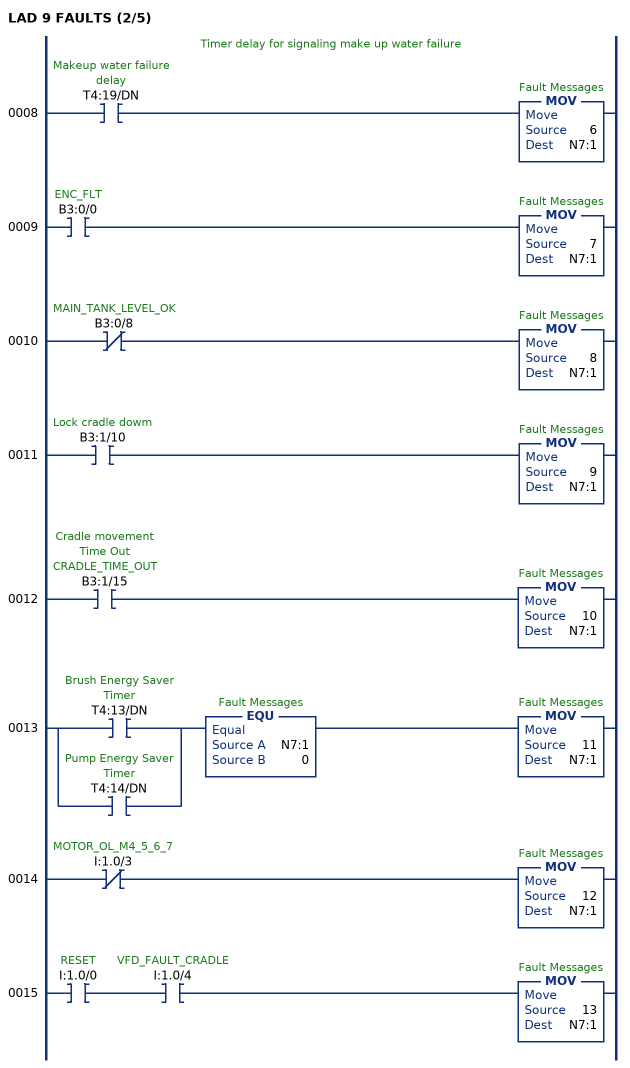
% Rung: 8 %
% Timer delay for signaling make up water failure %
SOR XIC T4:19/DN MOV 6 N7:1 EOR
%   T4:19  "Makeup water failure delay" %
%   N7:1  "Fault Messages" %
% Rung: 9 %
SOR XIC B3:0/0 MOV 7 N7:1 EOR
%   B3:0/0  ENC_FLT %
%   N7:1  "Fault Messages" %
% Rung: 10 %
SOR XIO B3:0/8 MOV 8 N7:1 EOR
%   B3:0/8  MAIN_TANK_LEVEL_OK %
%   N7:1  "Fault Messages" %
% Rung: 11 %
SOR XIC B3:1/10 MOV 9 N7:1 EOR
%   B3:1/10  "Lock cradle dowm" %
%   N7:1  "Fault Messages" %
% Rung: 12 %
SOR XIC B3:1/15 MOV 10 N7:1 EOR
%   B3:1/15  CRADLE_TIME_OUT  "Cradle movement Time Out" %
%   N7:1  "Fault Messages" %
% Rung: 13 %
SOR BST XIC T4:13/DN NXB XIC T4:14/DN BND EQU N7:1 0 MOV 11 N7:1 EOR
%   T4:13  "Brush Energy Saver Timer" %
%   T4:14  "Pump Energy Saver Timer" %
%   N7:1  "Fault Messages" %
% Rung: 14 %
SOR XIO I:1.0/3 MOV 12 N7:1 EOR
%   I:1.0/3  MOTOR_OL_M4_5_6_7 %
%   N7:1  "Fault Messages" %
% Rung: 15 %
SOR XIC I:1.0/0 XIC I:1.0/4 MOV 13 N7:1 EOR
%   I:1.0/0  RESET %
%   I:1.0/4  VFD_FAULT_CRADLE %
%   N7:1  "Fault Messages" %

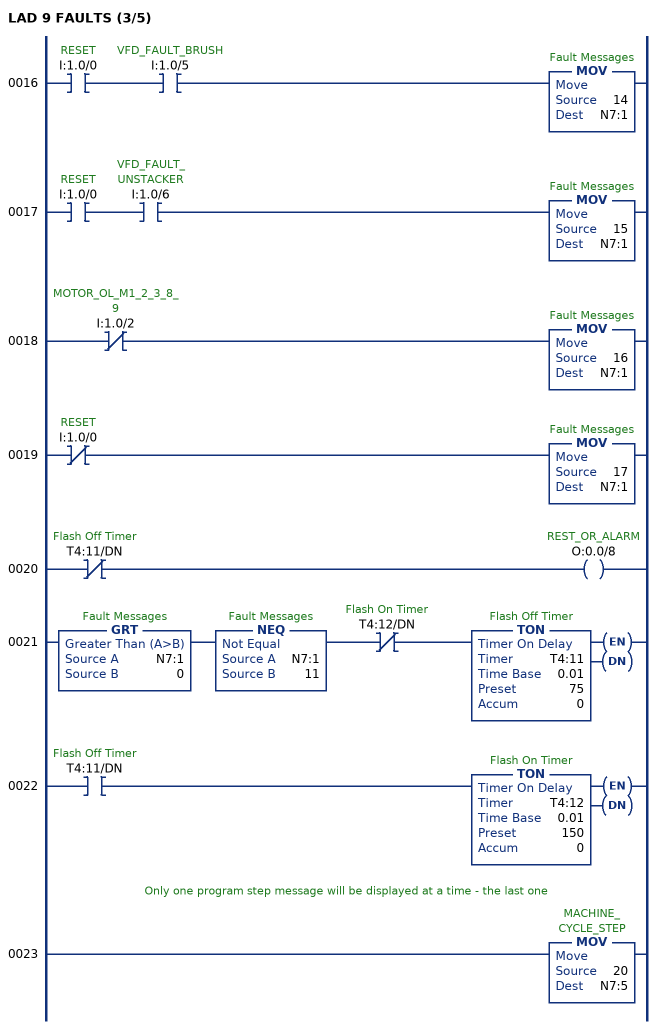
% Rung: 16 %
SOR XIC I:1.0/0 XIC I:1.0/5 MOV 14 N7:1 EOR
%   I:1.0/0  RESET %
%   I:1.0/5  VFD_FAULT_BRUSH %
%   N7:1  "Fault Messages" %
% Rung: 17 %
SOR XIC I:1.0/0 XIC I:1.0/6 MOV 15 N7:1 EOR
%   I:1.0/0  RESET %
%   I:1.0/6  VFD_FAULT_UNSTACKER %
%   N7:1  "Fault Messages" %
% Rung: 18 %
SOR XIO I:1.0/2 MOV 16 N7:1 EOR
%   I:1.0/2  MOTOR_OL_M1_2_3_8_9 %
%   N7:1  "Fault Messages" %
% Rung: 19 %
SOR XIO I:1.0/0 MOV 17 N7:1 EOR
%   I:1.0/0  RESET %
%   N7:1  "Fault Messages" %
% Rung: 20 %
SOR XIO T4:11/DN OTE O:0.0/8 EOR
%   T4:11  "Flash Off Timer" %
%   O:0.0/8  REST_OR_ALARM %
% Rung: 21 %
SOR GRT N7:1 0 NEQ N7:1 11 XIO T4:12/DN TON T4:11 0.01 75 0 EOR
%   N7:1  "Fault Messages" %
%   T4:12  "Flash On Timer" %
%   T4:11  "Flash Off Timer" %
% Rung: 22 %
SOR XIC T4:11/DN TON T4:12 0.01 150 0 EOR
%   T4:11  "Flash Off Timer" %
%   T4:12  "Flash On Timer" %
% Rung: 23 %
% Only one program step message will be displayed at a time - the last one %
SOR MOV 20 N7:5 EOR
%   N7:5  MACHINE_CYCLE_STEP %

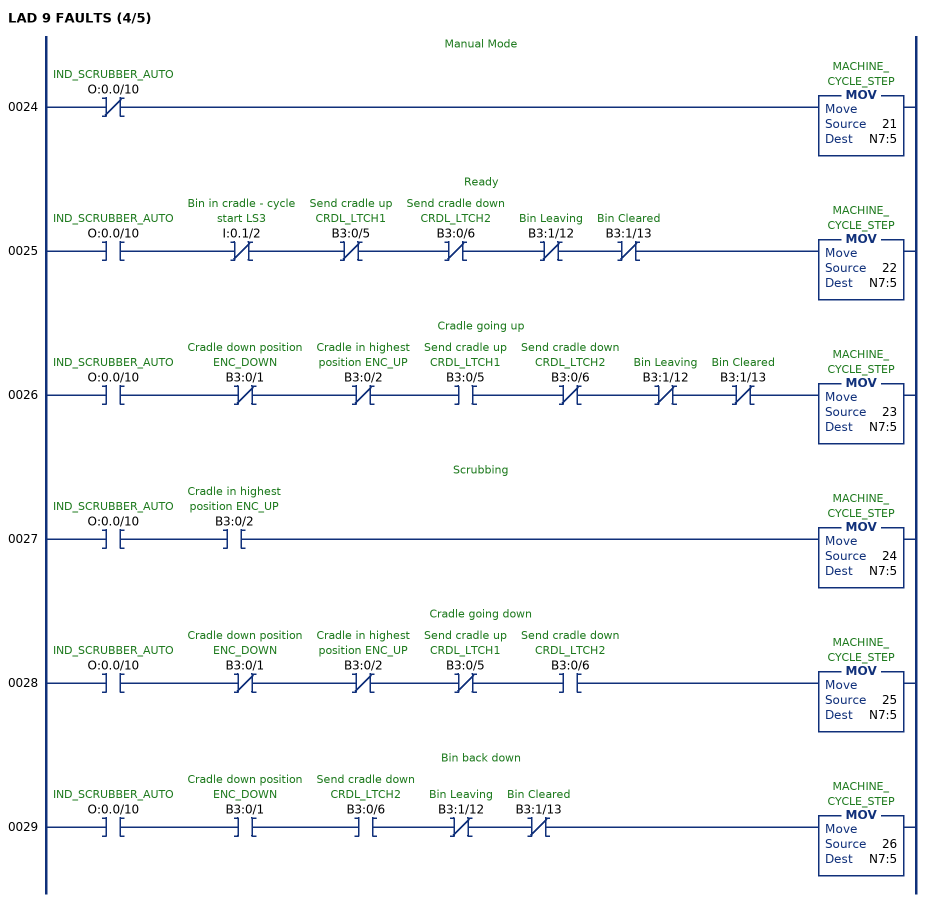
% Rung: 24 %
% Manual Mode %
SOR XIO O:0.0/10 MOV 21 N7:5 EOR
%   O:0.0/10  IND_SCRUBBER_AUTO %
%   N7:5  MACHINE_CYCLE_STEP %
% Rung: 25 %
% Ready %
SOR XIC O:0.0/10 XIO I:0.1/2 XIO B3:0/5 XIO B3:0/6 XIO B3:1/12 XIO B3:1/13 MOV 22 N7:5 EOR
%   O:0.0/10  IND_SCRUBBER_AUTO %
%   I:0.1/2  LS3  "Bin in cradle - cycle start" %
%   B3:0/5  CRDL_LTCH1  "Send cradle up" %
%   B3:0/6  CRDL_LTCH2  "Send cradle down" %
%   B3:1/12  "Bin Leaving" %
%   B3:1/13  "Bin Cleared" %
%   N7:5  MACHINE_CYCLE_STEP %
% Rung: 26 %
% Cradle going up %
SOR XIC O:0.0/10 XIO B3:0/1 XIO B3:0/2 XIC B3:0/5 XIO B3:0/6 XIO B3:1/12 XIO B3:1/13 MOV 23 N7:5 EOR
%   O:0.0/10  IND_SCRUBBER_AUTO %
%   B3:0/1  ENC_DOWN  "Cradle down position" %
%   B3:0/2  ENC_UP  "Cradle in highest position" %
%   B3:0/5  CRDL_LTCH1  "Send cradle up" %
%   B3:0/6  CRDL_LTCH2  "Send cradle down" %
%   B3:1/12  "Bin Leaving" %
%   B3:1/13  "Bin Cleared" %
%   N7:5  MACHINE_CYCLE_STEP %
% Rung: 27 %
% Scrubbing %
SOR XIC O:0.0/10 XIC B3:0/2 MOV 24 N7:5 EOR
%   O:0.0/10  IND_SCRUBBER_AUTO %
%   B3:0/2  ENC_UP  "Cradle in highest position" %
%   N7:5  MACHINE_CYCLE_STEP %
% Rung: 28 %
% Cradle going down %
SOR XIC O:0.0/10 XIO B3:0/1 XIO B3:0/2 XIO B3:0/5 XIC B3:0/6 MOV 25 N7:5 EOR
%   O:0.0/10  IND_SCRUBBER_AUTO %
%   B3:0/1  ENC_DOWN  "Cradle down position" %
%   B3:0/2  ENC_UP  "Cradle in highest position" %
%   B3:0/5  CRDL_LTCH1  "Send cradle up" %
%   B3:0/6  CRDL_LTCH2  "Send cradle down" %
%   N7:5  MACHINE_CYCLE_STEP %
% Rung: 29 %
% Bin back down %
SOR XIC O:0.0/10 XIC B3:0/1 XIC B3:0/6 XIO B3:1/12 XIO B3:1/13 MOV 26 N7:5 EOR
%   O:0.0/10  IND_SCRUBBER_AUTO %
%   B3:0/1  ENC_DOWN  "Cradle down position" %
%   B3:0/6  CRDL_LTCH2  "Send cradle down" %
%   B3:1/12  "Bin Leaving" %
%   B3:1/13  "Bin Cleared" %
%   N7:5  MACHINE_CYCLE_STEP %

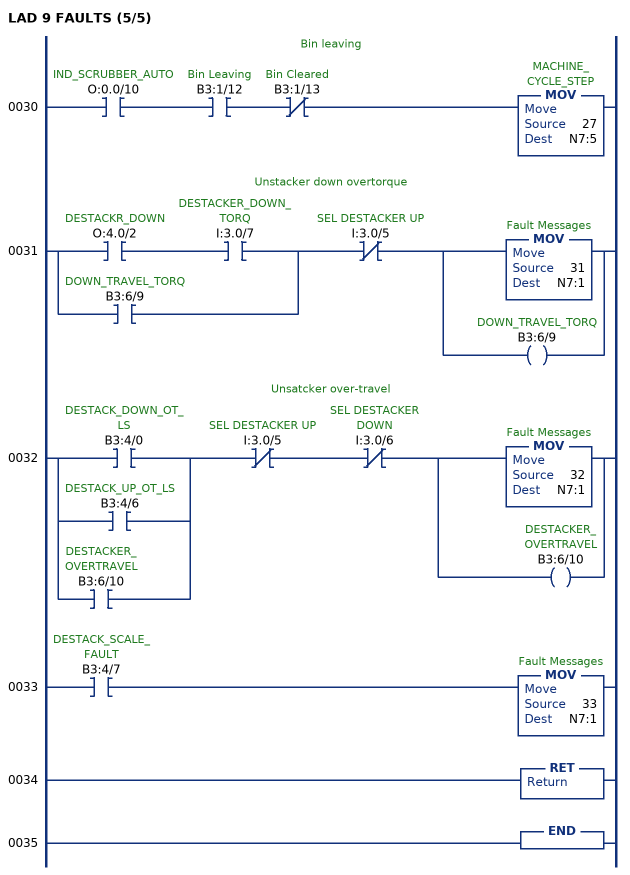
% Rung: 30 %
% Bin leaving %
SOR XIC O:0.0/10 XIC B3:1/12 XIO B3:1/13 MOV 27 N7:5 EOR
%   O:0.0/10  IND_SCRUBBER_AUTO %
%   B3:1/12  "Bin Leaving" %
%   B3:1/13  "Bin Cleared" %
%   N7:5  MACHINE_CYCLE_STEP %
% Rung: 31 %
% Unstacker down overtorque %
SOR BST XIC O:4.0/2 XIC I:3.0/7 NXB XIC B3:6/9 BND XIO I:3.0/5 BST MOV 31 N7:1 NXB OTE B3:6/9 BND EOR
%   O:4.0/2  DESTACKR_DOWN %
%   I:3.0/7  DESTACKER_DOWN_TORQ %
%   B3:6/9  DOWN_TRAVEL_TORQ %
%   I:3.0/5  "SEL DESTACKER UP" %
%   N7:1  "Fault Messages" %
% Rung: 32 %
% Unsatcker over-travel %
SOR BST BST XIC B3:4/0 NXB XIC B3:4/6 BND NXB XIC B3:6/10 BND XIO I:3.0/5 XIO I:3.0/6 BST MOV 32 N7:1 NXB OTE B3:6/10 BND EOR
%   B3:4/0  DESTACK_DOWN_OT_LS %
%   B3:4/6  DESTACK_UP_OT_LS %
%   B3:6/10  DESTACKER_OVERTRAVEL %
%   I:3.0/5  "SEL DESTACKER UP" %
%   I:3.0/6  "SEL DESTACKER DOWN" %
%   N7:1  "Fault Messages" %
% Rung: 33 %
SOR XIC B3:4/7 MOV 33 N7:1 EOR
%   B3:4/7  DESTACK_SCALE_FAULT %
%   N7:1  "Fault Messages" %
% Rung: 34 %
SOR RET EOR
% Rung: 35 %
SOR END EOR

LADDER 10 "SPARE"
